      uiState               := 20;
    END_IF
END_CASE
CASE uiState OF
  20:
    stState.bBusy           := FALSE;
    eStateActive            := eState + e_AxisFunction.AXIS_DONE;
    eStateExec	            := e_AxisFunction.AXIS_DONE;

  99:
    stState.bError          := TRUE;
    stState.bBusy           := FALSE;
    eStateActive            := eState + e_AxisFunction.ERROR;
    eStateExec	            := e_AxisFunction.ERROR;
END_CASE
END_ACTION

ACTION Axis_Halt:
CASE uiState OF
  0:
    eStateActive            := eState;
    stState.bBusy           := TRUE;
    stState.bReady          := FALSE;

    stMcOut                 := fbAxis.Halt(Execute        := FALSE,
                                           Deceleration	  := stCtrl.rDec, 
                                           Jerk					  := 100_000.0, 
                                           BufferMode		  := Tc2_MC2.MC_BufferMode.MC_Aborting);
    uiState                 := 10;
END_CASE
CASE uiState OF
  10:
    eStateActive            := eState + e_AxisFunction.AXIS_BUSY;
    eStateExec	            := e_AxisFunction.AXIS_BUSY;

    stMcOut                 := fbAxis.Halt(Execute        := TRUE,
                                           Deceleration	  := stCtrl.rDec, 
                                           Jerk					  := 100_000.0, 
                                           BufferMode		  := Tc2_MC2.MC_BufferMode.MC_Aborting);

    IF NOT stMcOut.Busy
    THEN
      IF stMcOut.Error
      THEN
        stState.uiErrorId		:= stMcOut.ErrorID;

        uiState             := 99;
  
      ELSIF stMcOut.Done
      THEN
        uiState             := 20;
      END_IF
      fbAxis.Halt(Execute         := FALSE,
                  Deceleration	  := stCtrl.rDec, 
                  Jerk					  := 100_000.0, 
                  BufferMode		  := Tc2_MC2.MC_BufferMode.MC_Aborting);
    END_IF
END_CASE
CASE uiState OF
  20:
    stState.bBusy           := FALSE;
    eStateActive            := eState + e_AxisFunction.AXIS_DONE;
    eStateExec		          := e_AxisFunction.AXIS_DONE;

  99:
    stState.bError          := TRUE;
    stState.bBusy           := FALSE;
    eStateActive            := eState + e_AxisFunction.ERROR;
    eStateExec	            := e_AxisFunction.ERROR;
END_CASE
END_ACTION

ACTION Axis_Home:
CASE uiState OF
  0:
    eStateActive            := eState;
    stState.bBusy           := TRUE;

    stMcOut                 := fbAxis.Home(Execute    := FALSE,
                                           Position		:= stHomingOptions.Position, 
                                           HomingMode	:= Tc2_MC2.MC_HomingMode.MC_ResetCalibration, 
                                           Options		:= stHomingOptions.Options);
    IF NOT bXenaxDrive
    THEN
      IF fbAxis.pAxisRef^.Status.Homed
      THEN
        uiState             := 10;
      ELSE
        uiState             := 15;
      END_IF
    ELSE
      uiState               := 100;
    END_IF
END_CASE
CASE uiState OF
  10:
    // always reset calibration to force a homing run of the axis
    eStateActive            := eState + e_AxisFunction.AXIS_BUSY;
    eStateExec	            := e_AxisFunction.AXIS_BUSY;

    stState.bReferenced     := FALSE;

    stMcOut                 := fbAxis.Home(Execute    := TRUE,
                                           Position		:= stHomingOptions.Position, 
                                           HomingMode	:= Tc2_MC2.MC_HomingMode.MC_ResetCalibration, 
                                           Options		:= stHomingOptions.Options);
    IF stMcOut.Done
    THEN
      stMcOut               := fbAxis.Home(Execute    := FALSE,
                                           Position		:= stHomingOptions.Position, 
                                           HomingMode	:= stHomingOptions.HomingMode, 
                                           Options		:= stHomingOptions.Options);

      IF (stHomingOptions.HomingMode = Tc2_MC2.MC_HomingMode.MC_Absolute)
      THEN
        uiState             := 20;
      ELSE
        uiState             := 15;	
      END_IF
    END_IF
END_CASE
CASE uiState OF
  15:
    stMcOut                 := fbAxis.Home(Execute    := TRUE,
                                           Position		:= stHomingOptions.Position, 
                                           HomingMode	:= stHomingOptions.HomingMode, 
                                           Options		:= stHomingOptions.Options);

    IF stMcOut.Done
    THEN
      stState.bReferenced   := fbAxis.pAxisRef^.Status.Homed;

      stMcOut               := fbAxis.Home(Execute    := FALSE,
                                           Position		:= stHomingOptions.Position, 
                                           HomingMode	:= stHomingOptions.HomingMode, 
                                           Options		:= stHomingOptions.Options);
      uiState               := 20;

    ELSIF stMcOut.Error
    THEN
      stState.uiErrorId		  := stMcOut.ErrorID;
      stMcOut               := fbAxis.Home(Execute    := FALSE,
                                           Position		:= stHomingOptions.Position, 
                                           HomingMode	:= stHomingOptions.HomingMode, 
                                           Options		:= stHomingOptions.Options);
      uiState               := 99;
    END_IF

  20:
    stState.bBusy           := FALSE;
    eStateActive            := eState + e_AxisFunction.AXIS_DONE;
    eStateExec	            := e_AxisFunction.AXIS_DONE;

  99:
    stState.bError          := TRUE;
    stState.bBusy           := FALSE;
    eStateActive            := eState + e_AxisFunction.ERROR;
    eStateExec	            := e_AxisFunction.ERROR;
END_CASE
CASE uiState OF
  // Xenax drive homing
  100:
    eStateActive            := eState + e_AxisFunction.AXIS_BUSY;
    stState.bReferenced 		:= FALSE;
    fbXenaxHoming.bExecute 	:= FALSE;

    uiState                 := 110;
END_CASE
CASE uiState OF
  110:
    fbXenaxHoming.bExecute  := TRUE;
    uiState                 := 120;

  120:
    IF fbXenaxHoming.Error
    THEN
      stState.uiErrorId     := fbXenaxHoming.ErrorId;
      uiState               := 99;

    ELSIF fbXenaxHoming.Done
    THEN
      stState.bReferenced 	:= TRUE;
      fbXenaxHoming.bExecute:= FALSE;

      uiState               := 20;
    END_IF
END_CASE
END_ACTION

ACTION Axis_Idle:
IF stState.bReady
THEN
  IF NOT fbAxis.pAxisRef^.Status.Error
  THEN
    stState.bError  := FALSE;
  END_IF
  eStateActive      := eState;
  eStateExec	      := e_AxisFunction.AXIS_DONE;
END_IF

IF NOT stState.bReady
THEN
  eStateActive := eState;
  eStateExec	 := e_AxisFunction.AXIS_BUSY;
END_IF
END_ACTION

ACTION Axis_Init:
(*
-------------------------------------------------------------------------------
	INIT 
  - check for fbAxis to startUp --> sAxisName chec
  - check for fbAxis StartUpError --> Axis_Reset() and try again

  - get encodertype and set output bSercosAxis
	- get Axis Params from NC
	- get manufacturer device name for detecting use of Xenax drive

-------------------------------------------------------------------------------
*)
CASE uiInitState OF

  0:
  stState.bError          := FALSE;
  isizeOut                := SIZEOF(stState);
  iSizeIn	                := SIZEOF(stCtrl);
  bSercosAxis             := FALSE;
  sAxisName               := fbAxis.NcAxisName;

  IF fbAxis.StartUpDone
  THEN
    stMsg.eType 				  := E_MessageType.eMessageInfo;
    stMsg.eDevice 			  := E_Device.Axis;
    stMsg.eSubdevice 		  := e_Subdevice.General;
    stMsg.iErrorNumber 	  := fbAxis.pAxisRef^.NcToPlc.AxisId;
    stMsg.sText					  := 'Init: ';
    stMsg.sText					  := Tc2_Standard.CONCAT(stMsg.sText, sAxisName);
    f_MessageSet(stMsg);

    uiInitState           := 40;
    bXenaxDrive				    := FALSE;
    bSercosAxis           := FALSE;

    fbCoeRead(Execute	    := FALSE,
              NetId       := fbAxis.pAxisRef^.ADS.NetId, 
              Axis        := fbAxis.pAxisRef^);

    IF (fbAxis.EncoderType <> 1)
    THEN
      uiInitState         := 10;
    END_IF

  ELSE
    IF (stMsg.sText <> 'startup')
    THEN
      stMsg.eType 				:= E_MessageType.eMessageInfo;
      stMsg.eDevice 			:= E_Device.Axis;
      stMsg.eSubdevice 		:= e_Subdevice.General;
      stMsg.iErrorNumber 	:= fbAxis.pAxisRef^.NcToPlc.AxisId;
      stMsg.sText					:= 'startup';
      f_MessageSet(stMsg);
    END_IF

    IF (fbAxis.StartUpError)
    THEN
      stMsg.eType 				:= E_MessageType.eMessageError;
      stMsg.eDevice 			:= E_Device.Axis;
      stMsg.eSubdevice 		:= e_Subdevice.General;
      stMsg.iErrorNumber 	:= fbAxis.pAxisRef^.NcToPlc.AxisId;
      stMsg.sText					:= 'InitError: ';

      f_MessageSet(stMsg);

      uiInitState         := 90;
    END_IF
  END_IF

  10:
    // get manufacturer device name in CoE
    fbCoeRead.Index 		  := 16#1008;
    fbCoeRead.SubIndex 	  := 0;
    fbCoeRead.pDstBuf		  := ADR(sDriveType);
    fbCoeRead.BufLen		  := SIZEOF(sDriveType);

    fbCoeRead(Execute	    := TRUE,
              NetId       := fbAxis.pAxisRef^.ADS.NetId, 
              Axis        := fbAxis.pAxisRef^);

    IF fbCoeRead.Busy
    THEN
      uiInitState         := 20;
    END_IF

  20:
    fbCoeRead(
              NetId       := fbAxis.pAxisRef^.ADS.NetId, 
              Axis        := fbAxis.pAxisRef^);

    IF (fbCoeRead.Error)
    THEN
      uiInitState         := 90;

    ELSIF NOT fbCoeRead.Busy
    THEN
      stState.bError 		  := FALSE;
      stState.uiErrorId   := 0;
      uiInitState         := 30;
    END_IF

  30:
    IF (fbAxis.EncoderType = 8) OR
       (fbAxis.EncoderType = 9)
    THEN
      bSercosAxis         := TRUE;

      stMsg.eType 				:= E_MessageType.eMessageInfo;
      stMsg.eDevice 			:= E_Device.Axis;
      stMsg.eSubdevice 		:= e_Subdevice.General;
      stMsg.iErrorNumber 	:= fbAxis.pAxisRef^.NcToPlc.AxisId;
      stMsg.sText					:= Tc2_Standard.CONCAT(stMsg.sText,',');
      stMsg.sText					:= Tc2_Standard.CONCAT(stMsg.sText, 'SERCOS');
      f_MessageSet(stMsg);
    END_IF

    // check manufacturer device name for identifier string
    IF (FIND(sDriveType, sXenax) <> 0)
    THEN
      bXenaxDrive         := TRUE;

      stMsg.eType 				:= E_MessageType.eMessageInfo;
      stMsg.eDevice 			:= E_Device.Axis;
      stMsg.eSubdevice 		:= e_Subdevice.General;
      stMsg.iErrorNumber 	:= fbAxis.pAxisRef^.NcToPlc.AxisId;
      stMsg.sText					:= Tc2_Standard.CONCAT(stMsg.sText,',');
      stMsg.sText					:= Tc2_Standard.CONCAT(stMsg.sText,sXenax);
      f_MessageSet(stMsg);
    END_IF
    uiInitState           := 40;

  40:
    eStateExec	          := e_AxisFunction.AXIS_DONE;
    eStateExecOld         := e_AxisFunction.AXIS_DONE;
    stMsg.eType 				  := E_MessageType.eMessageInfo;
    stMsg.eDevice 			  := E_Device.Axis;
    stMsg.eSubdevice 		  := e_Subdevice.General;
    stMsg.iErrorNumber 	  := fbAxis.pAxisRef^.NcToPlc.AxisId;
    stMsg.sText					  := Tc2_Standard.CONCAT(stMsg.sText, ': ');
    stMsg.sText					  := Tc2_Standard.CONCAT(stMsg.sText, TO_STRING(eStateExec));
    f_MessageSet(stMsg);
    uiInitState           := 100;

  90:
    stState.bError        := TRUE;
    uiState               := 0;
    uiInitState           := 91;

  91:
    Axis_Reset();
    IF (eStateExec = e_AxisFunction.AXIS_DONE)
    THEN
      stMsg.eType 				:= E_MessageType.eMessageInfo;
      stMsg.eDevice 			:= E_Device.Axis;
      stMsg.eSubdevice 		:= e_Subdevice.General;
      stMsg.iErrorNumber 	:= fbAxis.pAxisRef^.NcToPlc.AxisId;
      stMsg.sText					:= 'Init Axis_Reset: ';

      uiInitState         := 0;
    END_IF

  100:
    bInit                 := TRUE;
END_CASE
END_ACTION

ACTION Axis_Move_Buffer:
CASE uiState OF
  0:
    eStateActive            := eState;
    stState.bBusy           := TRUE;
    stState.bReady          := FALSE;

    stMcOut                 := fbAxis.MoveAbsolute(Enable       := FALSE,
                                                   Position		  := stCtrl.rSetPos, 
                                                   Velocity		  := stCtrl.rSetVelo, 
                                                   Acceleration := stCtrl.rAcc, 
                                                   Deceleration := stCtrl.rDec, 
                                                   Jerk				  := 0, 
                                                   BufferMode	      := stMotionOptions.eBufferMode,
                                                   fActivePosition  := stState.rSetPos,
                                                   eState           := eBufferState);

    uiState                 := 10;
END_CASE
CASE uiState OF
  10:
    eStateActive            := eState + e_AxisFunction.AXIS_BUSY;
    eStateExec              := e_AxisFunction.AXIS_BUSY;

    stMcOut                 := fbAxis.MoveAbsolute(Enable       := TRUE,
                                                   Position     := stCtrl.rSetPos, 
                                                   Velocity     := stCtrl.rSetVelo, 
                                                   Acceleration := stCtrl.rAcc, 
                                                   Deceleration := stCtrl.rDec, 
                                                   Jerk         := 0, 
                                                   BufferMode	      := stMotionOptions.eBufferMode,
                                                   fActivePosition  := stState.rSetPos,
                                                   eState           := eBufferState);

    IF stMcOut.Error
    THEN
      stState.uiErrorId     := stMcOut.ErrorID;
      uiState               := 99;

      stMcOut               := fbAxis.MoveAbsolute(Enable     := FALSE,
                                                   Position		  := stCtrl.rSetPos, 
                                                   Velocity		  := stCtrl.rSetVelo, 
                                                   Acceleration := stCtrl.rAcc, 
                                                   Deceleration := stCtrl.rDec, 
                                                   Jerk				  := 0, 
                                                   BufferMode	      := stMotionOptions.eBufferMode,
                                                   fActivePosition  := stState.rSetPos,
                                                   eState           := eBufferState);

    END_IF
END_CASE
CASE uiState OF
  99:
    stState.bError          := TRUE;
    stState.bBusy           := FALSE;
    eStateActive            := eState + e_AxisFunction.ERROR;
    eBufferState            :=
    eStateExec	            := e_AxisFunction.ERROR;
END_CASE
END_ACTION

ACTION Axis_Move_Buffer_Velocity:
CASE uiState OF
  0:
    eStateActive            := eState;
    stState.bBusy           := TRUE;
    stState.bReady          := FALSE;
    uiState                 := 5;
END_CASE

CASE uiState OF
  5:
    eStateActive            := eState + e_AxisFunction.AXIS_BUSY;
    eStateExec	            := e_AxisFunction.AXIS_BUSY;

    stMcOut                 := fbAxis.MoveVelocity(FALSE,
                                                   stCtrl.rSetVelo,
                                                   stCtrl.rAcc,
                                                   stCtrl.rDec,
                                                   100_000,
                                                   stCtrl.iDirection,
                                                   BufferMode       := Tc2_MC2.MC_BufferMode.MC_Aborting,
                                                   fActiveVelocity  := stState.rSetPos,
                                                   eState           := eBufferState);
    uiState                 := 10;
END_CASE
CASE uiState OF
  10:
    eStateActive            := eState + e_AxisFunction.AXIS_BUSY;
    eStateExec	            := e_AxisFunction.AXIS_BUSY;

    stMcOut                 := fbAxis.MoveVelocity(TRUE,
                                                   stCtrl.rSetVelo,
                                                   stCtrl.rAcc,
                                                   stCtrl.rDec,
                                                   100_000,
                                                   stCtrl.iDirection,
                                                   BufferMode       := Tc2_MC2.MC_BufferMode.MC_Aborting,
                                                   fActiveVelocity  := stState.rSetPos,
                                                   eState           := eBufferState);

    IF stMcOut.Error
    THEN
      stMcOut               := fbAxis.MoveVelocity(FALSE,
                                                   stCtrl.rSetVelo,
                                                   stCtrl.rAcc,
                                                   stCtrl.rDec,
                                                   100_000,
                                                   stCtrl.iDirection,
                                                   BufferMode       := Tc2_MC2.MC_BufferMode.MC_Aborting,
                                                   fActiveVelocity  := stState.rSetPos,
                                                   eState           := eBufferState);

      stState.uiErrorId		  := stMcOut.ErrorID;

      uiState               := 99;
    END_IF
END_CASE

CASE uiState OF
  99:
    stState.bError          := TRUE;
    stState.bBusy           := FALSE;
    eStateActive            := eState + e_AxisFunction.ERROR;
    eBufferState            :=
    eStateExec	            := e_AxisFunction.ERROR;
END_CASE
END_ACTION

ACTION Axis_Move_Pos:
CASE uiState OF
  0:
    eStateActive            := eState;
    stState.bBusy           := TRUE;

    rSetPos                 := stCtrl.rSetPos;
    stMcOut                 := fbAxis.MovePtP(Execute     := FALSE,
                                              Position		:= rSetPos, 
                                              Velocity		:= stCtrl.rSetVelo, 
                                              Acceleration:= stCtrl.rAcc, 
                                              Deceleration:= stCtrl.rDec, 
                                              Jerk				:= 0);

    uiState                 := 10;
END_CASE
CASE uiState OF
  10:
    eStateActive            := eState + e_AxisFunction.AXIS_BUSY;
    eStateExec	            := e_AxisFunction.AXIS_BUSY;

    stMcOut                 := fbAxis.MovePtP(Execute     := TRUE,
                                              Position		:= rSetPos, 
                                              Velocity		:= stCtrl.rSetVelo, 
                                              Acceleration:= stCtrl.rAcc, 
                                              Deceleration:= stCtrl.rDec, 
                                              Jerk				:= 0); //default

    IF stMcOut.Done OR 
       stMcOut.Error
    THEN
      IF stMcOut.Done
      THEN
        uiState             := 11;
      END_IF
      IF stMcOut.Error
      THEN
        stState.uiErrorId		:= stMcOut.ErrorID;
        uiState             := 99;
      END_IF

      stMcOut               := fbAxis.MovePtP(Execute     := FALSE,
                                              Position		:= rSetPos, 
                                              Velocity		:= stCtrl.rSetVelo, 
                                              Acceleration:= stCtrl.rAcc, 
                                              Deceleration:= stCtrl.rDec, 
                                              Jerk				:= 0);
    END_IF
END_CASE
CASE uiState OF
  11:
    IF stState.bInTarget
    THEN
      uiState               := 20;
    END_IF
END_CASE
CASE uiState OF
  20:
    stState.bBusy           := FALSE;
    eStateActive            := eState + e_AxisFunction.AXIS_DONE;
    eStateExec	            := e_AxisFunction.AXIS_DONE;

  99:
    stState.bError          := TRUE;
    stState.bBusy           := FALSE;
    eStateActive            := eState + e_AxisFunction.ERROR;
    eStateExec              := e_AxisFunction.ERROR;
END_CASE
END_ACTION

ACTION Axis_Move_Velo:
CASE uiState OF
  0:
    eStateActive            := eState;
    stState.bBusy           := TRUE;
    stState.bReady          := FALSE;
    uiState := 5;
END_CASE

CASE uiState OF
  5:
    eStateActive            := eState + e_AxisFunction.AXIS_BUSY;
    eStateExec	            := e_AxisFunction.AXIS_BUSY;

    stMcOut                 := fbAxis.MoveVelocity(FALSE,
                                                   stCtrl.rSetVelo,
                                                   stCtrl.rAcc,
                                                   stCtrl.rDec,
                                                   100_000,
                                                   stCtrl.iDirection,
                                                   BufferMode       := Tc2_MC2.MC_BufferMode.MC_Aborting,
                                                   fActiveVelocity  := stState.rSetPos,
                                                   eState           := eBufferState);

    uiState                 := 10;
END_CASE
CASE uiState OF
  10:
    eStateActive            := eState + e_AxisFunction.AXIS_BUSY;
    eStateExec	            := e_AxisFunction.AXIS_BUSY;

    stMcOut                 := fbAxis.MoveVelocity(TRUE,
                                                   stCtrl.rSetVelo,
                                                   stCtrl.rAcc,
                                                   stCtrl.rDec,
                                                   100_000,
                                                   stCtrl.iDirection,
                                                   BufferMode       := Tc2_MC2.MC_BufferMode.MC_Aborting,
                                                   fActiveVelocity  := stState.rSetPos,
                                                   eState           := eBufferState);

    IF stMcOut.Error
    THEN
      stMcOut               := fbAxis.MoveVelocity(FALSE,
                                                   stCtrl.rSetVelo,
                                                   stCtrl.rAcc,
                                                   stCtrl.rDec,
                                                   100_000,
                                                   stCtrl.iDirection,
                                                   BufferMode       := Tc2_MC2.MC_BufferMode.MC_Aborting,
                                                   fActiveVelocity  := stState.rSetPos,
                                                   eState           := eBufferState);

      stState.uiErrorId     := stMcOut.ErrorID;

      uiState               := 99;

    ELSIF stMcOut.Done
    THEN
      stMcOut               := fbAxis.MoveVelocity(FALSE,
                                                   stCtrl.rSetVelo,
                                                   stCtrl.rAcc,
                                                   stCtrl.rDec,
                                                   100_000,
                                                   stCtrl.iDirection,
                                                   BufferMode       := Tc2_MC2.MC_BufferMode.MC_Aborting,
                                                   fActiveVelocity  := stState.rSetPos,
                                                   eState           := eBufferState);

      uiState               := 20;
    END_IF
END_CASE

CASE uiState OF
  20:
    stState.bBusy           := FALSE;
    eStateActive            := eState + e_AxisFunction.AXIS_DONE;
    eStateExec              := e_AxisFunction.AXIS_DONE;

  99:
    stState.bError          := TRUE;
    stState.bBusy           := FALSE;
    eStateActive            := eState + e_AxisFunction.ERROR;
    eStateExec              := e_AxisFunction.ERROR;
END_CASE
END_ACTION

ACTION Axis_Parameter:
CASE uiState OF
  0:
    eStateActive            := eState;

    tonWaitSeq(IN           := FALSE);

    IF stNcParameter.bRead
    THEN
      stState.bBusy         := TRUE;
      stMcOut               := fbAxis.ReadParameter(FALSE,stNcParameter.ParameterNumber);
      uiState               := 10;

    ELSIF stNcParameter.bWrite
    THEN
      stState.bBusy         := TRUE;
      stMcOut               := fbAxis.WriteParameter(FALSE, stNcParameter.ParameterNumber, stNcParameter.rValueWrite);
      uiState               := 11;
    END_IF

  10:
    eStateActive            := eState + e_AxisFunction.AXIS_BUSY;
    eStateExec              := e_AxisFunction.AXIS_BUSY;

    tonWaitSeq(IN           := TRUE, 
               PT           := T#50MS);

    stMcOut                 := fbAxis.ReadParameter(TRUE,stNcParameter.ParameterNumber);

    IF stMcOut.Done AND 
       tonWaitSeq.Q
    THEN
      stNcParameter.rValueRead  := LREAL_TO_REAL(fbAxis.ReadParamValue);
      stMcOut                   := fbAxis.ReadParameter(FALSE,stNcParameter.ParameterNumber);

      uiState               := 20;
    END_IF

  11:
    eStateActive            := eState + e_AxisFunction.AXIS_BUSY;
    eStateExec              := e_AxisFunction.AXIS_BUSY;

    tonWaitSeq(IN           := TRUE, 
               PT           := T#50MS);

    stMcOut                 := fbAxis.WriteParameter(TRUE, stNcParameter.ParameterNumber, stNcParameter.rValueWrite);

    IF stMcOut.Done AND 
       tonWaitSeq.Q
    THEN
      IF fbAxis.LocalParameterReload()
      THEN
        stMcOut             := fbAxis.WriteParameter(FALSE, stNcParameter.ParameterNumber, stNcParameter.rValueWrite);
        uiState             := 20;
      END_IF
    END_IF

  20:
    stState.bBusy           := FALSE;
    eStateActive            := eState + e_AxisFunction.AXIS_DONE;
    eStateExec              := e_AxisFunction.AXIS_DONE;
END_CASE
END_ACTION

ACTION Axis_Reset:
CASE uiState OF
  0:
    eStateActive            := eState;
    stState.bBusy           := TRUE;
    stState.bReady          := FALSE;
    stState.bTimeout        := FALSE;
    stMcOut                 := fbAxis.ErrorReset(FALSE);

    uiState                 := 10;
END_CASE
CASE uiState OF
  10:
    eStateActive            := eState + e_AxisFunction.AXIS_BUSY;
    eStateExec              := e_AxisFunction.AXIS_BUSY;
    stMcOut                 := fbAxis.ErrorReset(TRUE);

    IF stMcOut.Done
    THEN
      stState.bError        := FALSE;
      stState.uiErrorId     := 0;
      stMcOut               := fbAxis.ErrorReset(FALSE);
      uiState               := 20;

    ELSIF stMcOut.Error
    THEN
      stState.uiErrorId		  := stMcOut.ErrorID;
      uiState               := 99;
    END_IF
END_CASE
CASE uiState OF
  20:
    fbResetSercos(bExecute	:= FALSE);

    IF fbAxis.pAxisRef^.Status.DriveDeviceError AND
       bSercosAxis
    THEN
      tonTimeout(IN         := FALSE, 
                 PT         := tUpdate);

      uiState               := 30;
    ELSE
      uiState               := 40;
    END_IF

END_CASE
CASE uiState OF
  30:
    tonTimeout(IN           := TRUE, 
               PT           := tUpdate);

    fbResetSercos(bExecute	:= TRUE, 
                  p_AxisRef	:= ADR(fbAxis._AxisRef), stMcOutput=> );

    IF tonTimeout.Q
    THEN
      uiState               := 0;
    ELSE
      IF NOT fbAxis.pAxisRef^.Status.DriveDeviceError
      THEN
        tonTimeout(IN       := FALSE, 
                   PT       := tUpdate);

        uiState             := 40;
      END_IF
    END_IF
END_CASE
CASE uiState OF
  40:
    stState.bBusy           := FALSE;
    eStateActive            := eState + e_AxisFunction.AXIS_DONE;
    eStateExec              := e_AxisFunction.AXIS_DONE;


  99:
    stState.bError          := TRUE;
    stState.bBusy           := FALSE;
    eStateActive            := eState + e_AxisFunction.ERROR;
    eStateExec              := e_AxisFunction.ERROR;
END_CASE
END_ACTION

ACTION Axis_Reset_SS1:
CASE uiState OF
  0:
    eStateActive            := eState;
    stState.bBusy           := TRUE;
    stState.bReady          := FALSE;
    stState.bTimeout        := FALSE;
    stMcOut                 := fbAxis.ErrorReset(FALSE);

    uiState                 := 10;
END_CASE
CASE uiState OF
  10:
    eStateActive            := eState + e_AxisFunction.AXIS_BUSY;
    eStateExec              := e_AxisFunction.AXIS_BUSY;
    stMcOut                 := fbAxis.ErrorReset(TRUE);

    IF NOT stMcOut.Busy
    THEN
      stMcOut               := fbAxis.ErrorReset(FALSE);
      uiState               := 20;

    ELSIF stMcOut.Error
    THEN
      stState.uiErrorId		  := stMcOut.ErrorID;
      uiState               := 99;
    END_IF
END_CASE
CASE uiState OF
  20:
    fbResetSercos(bExecute	:= FALSE);

    IF fbAxis.pAxisRef^.Status.DriveDeviceError AND
       bSercosAxis
    THEN
      tonTimeout(IN         := FALSE, 
                 PT         := tUpdate);

      uiState               := 30;
    ELSE
      uiState               := 40;
    END_IF

END_CASE
CASE uiState OF
  30:
    tonTimeout(IN           := TRUE, 
               PT           := tUpdate);

    fbResetSercos(bExecute	:= TRUE, 
                  p_AxisRef	:= ADR(fbAxis._AxisRef), stMcOutput=> );

    IF tonTimeout.Q
    THEN
      uiState               := 0;
    ELSE
      IF NOT fbAxis.pAxisRef^.Status.DriveDeviceError
      THEN
        tonTimeout(IN       := FALSE, 
                   PT       := tUpdate);

        uiState             := 40;
      END_IF
    END_IF
END_CASE
CASE uiState OF
  40:
    stState.bBusy           := FALSE;
    eStateActive            := eState + e_AxisFunction.AXIS_DONE;
    eStateExec              := e_AxisFunction.AXIS_DONE;


  99:
    stState.bError          := TRUE;
    stState.bBusy           := FALSE;
    eStateActive            := eState + e_AxisFunction.ERROR;
    eStateExec              := e_AxisFunction.ERROR;
END_CASE
END_ACTION

ACTION Axis_Stop:
CASE uiState OF
  0:
    eStateActive            := eState;
    stState.bBusy           := TRUE;
    stState.bReady          := FALSE;

    stMcOut                 := fbAxis.Stop(FALSE);
    uiState                 := 10;
END_CASE
CASE uiState OF
  10:
    eStateActive            := eState + e_AxisFunction.AXIS_BUSY;
    eStateExec              := e_AxisFunction.AXIS_BUSY;

    stMcOut                 := fbAxis.Stop(TRUE);

    IF stMcOut.Error
    THEN
      stState.uiErrorId		  := stMcOut.ErrorID;
      stMcOut               := fbAxis.Stop(FALSE);
      uiState               := 99;

    ELSIF stMcOut.Done
    THEN
      stMcOut               := fbAxis.Stop(FALSE);
      uiState               := 20;
    END_IF
END_CASE
CASE uiState OF
  20:
    stState.bBusy           := FALSE;

    eStateActive            := eState + e_AxisFunction.AXIS_DONE;
    eStateExec              := e_AxisFunction.AXIS_DONE;

  99:
    stState.bError          := TRUE;
    stState.bBusy           := FALSE;

    eStateActive            := eState + e_AxisFunction.ERROR;
    eStateExec              := e_AxisFunction.ERROR;
END_CASE
END_ACTION

ACTION Axis_Stop_SS1:

eStateActive                := e_AxisFunction.AXIS_SS1_STOP + e_AxisFunction.AXIS_BUSY;
eStateExec	                := e_AxisFunction.AXIS_BUSY;

stState.bBusy               := TRUE;
stState.bReady              := FALSE;

CASE uiStateSS1 OF
   0:
    IF fbAxis.Enable
    THEN
      uiStateSS1            := 10;
    ELSE
      uiStateSS1            := 100;
    END_IF
END_CASE
CASE uiStateSS1 OF
  10:
    fbAxis.Stop(FALSE);
    uiStateSS1              := 20;
END_CASE
CASE uiStateSS1 OF
  20:
    fbAxis.Stop(TRUE);
    IF fbAxis._AxisRef.Status.NotMoving
    THEN
      uiStateSS1            := 100;
    END_IF
END_CASE
CASE uiStateSS1 OF
  100:
    uiStateSS1              := 0;
    fbAxis.Enable           := FALSE;
    stState.bBusy           := FALSE;
    eStateActive            := e_AxisFunction.AXIS_SS1_STOP + e_AxisFunction.AXIS_DONE;
    eStateExec              := e_AxisFunction.AXIS_DONE;
END_CASE
END_ACTION

ACTION Axis_WriteBufferMode:

CASE uiState OF
  0:
    eStateActive            := eState;
    stState.bBusy           := TRUE;
    stState.bReady          := FALSE;

    uiState                 := 10;
END_CASE
CASE uiState OF
  10:
    eStateActive            := eState + e_AxisFunction.AXIS_BUSY;
    eStateExec	            := e_AxisFunction.AXIS_BUSY;

END_CASE
CASE uiState OF
  20:
    stState.bBusy           := FALSE;
    eStateActive            := eState + e_AxisFunction.AXIS_DONE;
    eStateExec	            := e_AxisFunction.AXIS_DONE;

  99:
    stState.bError          := TRUE;
    stState.bBusy           := FALSE;
    eStateActive            := eState + e_AxisFunction.ERROR;
    eStateExec	            := e_AxisFunction.ERROR;
END_CASE
END_ACTION

PROPERTY MasterAxis1 : POINTER TO Tc2_MC2.AXIS_REF
GET
MasterAxis1 := _pAxis1;
END_GET
SET
IF MasterAxis1 = 0 THEN
	_pAxis1 := ADR(st_AxisREF_Dummy);
ELSE
	_pAxis1 := MasterAxis1;	
END_IF
END_SET
END_PROPERTY

PROPERTY MasterAxis2 : POINTER TO Tc2_MC2.AXIS_REF
GET
MasterAxis2 := _pAxis2;
END_GET
SET
IF MasterAxis2 = 0 THEN
	_pAxis2 := ADR(st_AxisREF_Dummy);
ELSE
	_pAxis2 := MasterAxis2;	
END_IF
END_SET
END_PROPERTY

PROPERTY MasterAxis3 : POINTER TO Tc2_MC2.AXIS_REF
GET
MasterAxis3 := _pAxis3;
END_GET
SET
IF MasterAxis3 = 0 THEN
	_pAxis3 := ADR(st_AxisREF_Dummy);
ELSE
	_pAxis3 := MasterAxis3;	
END_IF
END_SET
END_PROPERTY

PROPERTY MasterAxis4 : POINTER TO Tc2_MC2.AXIS_REF
GET
MasterAxis4 := _pAxis4;
END_GET
SET
IF MasterAxis4 = 0 THEN
	_pAxis4 := ADR(st_AxisREF_Dummy);
ELSE
	_pAxis4 := MasterAxis4;	
END_IF
END_SET
END_PROPERTY

PROPERTY PUBLIC StatusCompact : ST_AxisStatusCompact
GET


_stStatusCompact.Error                := fbAxis.pAxisRef^.Status.Error;
(* PLCopen motion control statemachine states: *)
_stStatusCompact.ErrorStop            := fbAxis.pAxisRef^.Status.ErrorStop;
_stStatusCompact.Disabled             := fbAxis.pAxisRef^.Status.Disabled;
_stStatusCompact.Stopping             := fbAxis.pAxisRef^.Status.Stopping;

_stStatusCompact.StandStill           := fbAxis.pAxisRef^.Status.StandStill;
_stStatusCompact.DiscreteMotion       := fbAxis.pAxisRef^.Status.DiscreteMotion;
_stStatusCompact.ContinuousMotion     := fbAxis.pAxisRef^.Status.ContinuousMotion; 
_stStatusCompact.SynchronizedMotion   := fbAxis.pAxisRef^.Status.SynchronizedMotion;

_stStatusCompact.Homing               := fbAxis.pAxisRef^.Status.Homing;

(* additional status - (PLCopen definition)*)
_stStatusCompact.ConstantVelocity     := fbAxis.pAxisRef^.Status.ConstantVelocity; 
_stStatusCompact.Accelerating         := fbAxis.pAxisRef^.Status.Accelerating;
_stStatusCompact.Decelerating         := fbAxis.pAxisRef^.Status.Decelerating;

(* Axis.NcToPlc.StateDWord *)
_stStatusCompact.Operational          := fbAxis.pAxisRef^.Status.Operational; 
_stStatusCompact.ControlLoopClosed    := fbAxis.pAxisRef^.Status.ControlLoopClosed;
_stStatusCompact.HasJob               := fbAxis.pAxisRef^.Status.HasJob; 
_stStatusCompact.HasBeenStopped       := fbAxis.pAxisRef^.Status.HasBeenStopped; 
_stStatusCompact.NewTargetPosition    := fbAxis.pAxisRef^.Status.NewTargetPosition;
_stStatusCompact.InPositionArea       := fbAxis.pAxisRef^.Status.InPositionArea; 
_stStatusCompact.InTargetPosition     := fbAxis.pAxisRef^.Status.InTargetPosition; 

_stStatusCompact.Homed                := fbAxis.pAxisRef^.Status.Homed; 
_stStatusCompact.HomingBusy           := fbAxis.pAxisRef^.Status.HomingBusy; 
_stStatusCompact.MotionCommandsLocked := fbAxis.pAxisRef^.Status.MotionCommandsLocked;
_stStatusCompact.SoftLimitMinExceeded := fbAxis.pAxisRef^.Status.SoftLimitMinExceeded;
_stStatusCompact.SoftLimitMaxExceeded := fbAxis.pAxisRef^.Status.SoftLimitMaxExceeded;

_stStatusCompact.Moving               := fbAxis.pAxisRef^.Status.Moving; 
_stStatusCompact.PositiveDirection    := fbAxis.pAxisRef^.Status.PositiveDirection; 
_stStatusCompact.NegativeDirection    := fbAxis.pAxisRef^.Status.NegativeDirection; 
_stStatusCompact.NotMoving            := fbAxis.pAxisRef^.Status.NotMoving; 
_stStatusCompact.Compensating         := fbAxis.pAxisRef^.Status.Compensating;

_stStatusCompact.ExtSetPointGenEnabled:= fbAxis.pAxisRef^.Status.ExtSetPointGenEnabled; 
_stStatusCompact.ExternalLatchValid   := fbAxis.pAxisRef^.Status.ExternalLatchValid; 
_stStatusCompact.CamDataQueued        := fbAxis.pAxisRef^.Status.CamDataQueued; 
_stStatusCompact.CamTableQueued       := fbAxis.pAxisRef^.Status.CamTableQueued; 
_stStatusCompact.CamScalingPending    := fbAxis.pAxisRef^.Status.CamScalingPending; 
_stStatusCompact.CmdBuffered          := fbAxis.pAxisRef^.Status.CmdBuffered; 
_stStatusCompact.PTPmode              := fbAxis.pAxisRef^.Status.PTPmode; 
_stStatusCompact.DriveDeviceError     := fbAxis.pAxisRef^.Status.DriveDeviceError; 
_stStatusCompact.IoDataInvalid        := fbAxis.pAxisRef^.Status.IoDataInvalid; 

(* Axis.NcToPlc.CoupleState *)
_stStatusCompact.Coupled              := fbAxis.pAxisRef^.Status.Coupled;

StatusCompact := _stStatusCompact;
END_GET
END_PROPERTY

PROPERTY stCam : ST_CamIn
GET
stCam := _stCamIn;
END_GET
SET
_stCamIn := stCam;

IF NOT IsFinite(F_Real(_stCamIn.MasterOffset))
THEN
  _stCamIn.MasterOffset := 0.0;
END_IF

IF NOT IsFinite(F_Real(_stCamIn.SlaveOffset))
THEN
  _stCamIn.SlaveOffset := 0.0;
END_IF

IF NOT IsFinite(F_Real(_stCamIn.MasterScaling))
THEN
  _stCamIn.MasterScaling := 0.0;
END_IF

IF NOT IsFinite(F_Real(_stCamIn.SlaveScaling))
THEN
  _stCamIn.SlaveScaling := 0.0;
END_IF
END_SET
END_PROPERTY

PROPERTY stGear : ST_GearIn
GET
stGear := _stGearIn;
END_GET
SET
_stGearIn := stGear;

IF NOT IsFinite(F_Real(_stGearIn.Acceleration))
THEN
  _stGearIn.Acceleration := 0.0;
END_IF

IF NOT IsFinite(F_Real(_stGearIn.Deceleration))
THEN
  _stGearIn.Deceleration := 0.0;
END_IF

IF NOT IsFinite(F_Real(_stGearIn.Jerk))
THEN
  _stGearIn.Jerk := 0.0;
END_IF

IF NOT IsFinite(F_Real(_stGearIn.RatioNumerator))
THEN
  _stGearIn.RatioNumerator := 0.0;
END_IF
END_SET
END_PROPERTY

PROPERTY stGearMultiMaster : ST_GearInMultiMaster
GET
stGearMultiMaster := _stGearInMultiMaster;
END_GET
SET
_stGearInMultiMaster := stGearMultiMaster;

IF NOT IsFinite(F_Real(_stGearInMultiMaster.Acceleration))
THEN
  _stGearInMultiMaster.Acceleration := 0.0;
END_IF

IF NOT IsFinite(F_Real(_stGearInMultiMaster.Deceleration))
THEN
  _stGearInMultiMaster.Deceleration := 0.0;
END_IF

IF NOT IsFinite(F_Real(_stGearInMultiMaster.Jerk))
THEN
  _stGearInMultiMaster.Jerk := 0.0;
END_IF

IF NOT IsFinite(F_Real(_stGearInMultiMaster.GearRatio1))
THEN
  _stGearInMultiMaster.GearRatio1 := 0.0;
END_IF

IF NOT IsFinite(F_Real(_stGearInMultiMaster.GearRatio2))
THEN
  _stGearInMultiMaster.GearRatio2 := 0.0;
END_IF

IF NOT IsFinite(F_Real(_stGearInMultiMaster.GearRatio3))
THEN
  _stGearInMultiMaster.GearRatio3 := 0.0;
END_IF

IF NOT IsFinite(F_Real(_stGearInMultiMaster.GearRatio4))
THEN
  _stGearInMultiMaster.GearRatio4 := 0.0;
END_IF
END_SET
END_PROPERTY

END_FUNCTION_BLOCK

// ---- POUs/NC_AXIS/FB_McPtpAxis.TcPOU
FUNCTION_BLOCK FB_McPtpAxis IMPLEMENTS I_McAxis
VAR
  _AxisRef                    : Tc2_MC2.AXIS_REF;
  pCalibrationCam             : POINTER TO BOOL;
  bConnectProps2NcParams      : BOOL := TRUE;
  stDefaultAcceleration       : ST_Param;
  stDefaultDeceleration       : ST_Param;
  stDefaultJerk               : ST_Param;
  fDefaultVelocity            : LREAL;

  stHomingSearchVelo          : ST_Param;
  stHomingVelo                : ST_Param;
  stMaxAcceleration           : ST_Param;
  stMaxDeceleration           : ST_Param;
  stMaxVelocity               : ST_Param;
  stTargetPositionWindow      : ST_Param;


  stSwPosLimitNegative        : ST_Param;
  stSwPosLimitNegativeActive  : ST_BoolParam;
  stSwPosLimitPositive        : ST_Param;
  stSwPosLimitPositiveActive  : ST_BoolParam;
  fReadParamValue             : LREAL;
  stAxisStatus                : Tc2_MC2.ST_AxisStatus;

  // name and encoder type are read by ADSREAD instance from NC
  stAxisName                  : STRING(30) := 'NO NAME'; // AxisName is limited to 30 chars, IdxGrp := 4000 + _AxisRef.NcToPlc.AxisId, IdxOffs := 16#02
  stEncoderType               : STRING(30) := 'NO TYPE';
  eEncoderType                : E_AxisEncoderType;
  
  // Motion Control FB Instances
  fbPower                     : MC_Power;
  fbReset                     : MC_Reset;
  fbHalt                      : MC_Halt;
  fbStop                      : MC_Stop;
  fbHome                      : MC_Home;
  fbJog                       : MC_Jog;

  fbReadParameter             : MC_ReadParameter;
  fbWriteParameter            : Tc2_MC2.MC_WriteParameter;
  fbMoveVelocity1             : MC_MoveVelocity;
  fbMoveVelocity2             : MC_MoveVelocity;
  fbMoveAbsolute1             : MC_MoveAbsolute;
  fbMoveAbsolute2             : MC_MoveAbsolute;
  fbMoveEndless               : Tc2_MC2.MC_MoveContinuousAbsolute;

  // ADS read instance for reading startup information from NC
  fbADSRead                   : ADSREAD;

  // private vars for Methode Params
  stHaltParams                : ST_HaltParams;
  stHomeParams                : ST_HomeParams;
  stJogParams                 : ST_JogParams;
  stMoveAbsParams             : ST_MoveAbsParams;
  stMoveVeloParams            : ST_MoveVeloParams;
  stReadParamParams           : ST_ReadParamParams; 
  stStopParams                : ST_StopParams;
  stWriteParamParams          : ST_WriteParamParams;

  // local message list for online debug
  stMsg                       : ST_Message;
  atMsg                       : ARRAY[1..MAX_MSG_INTERN] OF ST_Message;
  itMsg                       : DINT := 1;

  // startup states for getting ADS information from NC
  _nStartUpErrorState,
  _nStartUp                   : DINT := 0;

  _bStartUpError,
  _bStartUp                   : BOOL;

  _uiEncoderType              : UDINT;

  _rCycleTime                 : LREAL;
  fbGetCurTaskIndex           : Tc2_System.GETCURTASKINDEX;

END_VAR
VAR CONSTANT
  MAX_MSG_INTERN              : DINT := 10;
END_VAR

fbPower(Axis:= _AxisRef);
_AxisRef();

IF NOT _bStartUp
THEN
  CASE _nStartUp OF
    0:
      // wait for cyclic data to be valid / connected
      IF (_AxisRef.NcToPlc.AxisId > 0)
      THEN
        fbADSRead(NETID       := '', 
                  PORT        := 501, 
                  IDXGRP      := (16#5000 + _AxisRef.NcToPlc.AxisId), 
                  IDXOFFS     := 16#00000003, // offset for encoder type
                  LEN         := SIZEOF(_uiEncoderType), 
                  DESTADDR    := ADR(_uiEncoderType),
                  TMOUT       := T#200MS,
                  READ        := FALSE);

        // clear required ADS information
        stAxisName            := 'NO NAME';
        _uiEncoderType        :=  0;
        _nStartUpErrorState   :=  0;  // debug
        _nStartUp             := 10;
      END_IF

  10:
    fbADSRead(NETID           := '', 
              PORT            := 501, 
              IDXGRP          := (16#5000 + _AxisRef.NcToPlc.AxisId), 
              IDXOFFS         := 16#00000003, // offset for encoder type
              LEN             := SIZEOF(_uiEncoderType), 
              DESTADDR        := ADR(_uiEncoderType),
              READ            := TRUE);

    IF fbADSRead.ERR
    THEN
      stMsg.eType             := E_MessageType.eMessageError;
      stMsg.eDevice           := e_Device.Axis;
      stMsg.eSubdevice        := e_Subdevice.General;
      stMsg.iErrorNumber      := fbAdsRead.ERRID;
      stMsg.sText             := 'StartUp Ads Error Read Encoder Type';

      MsgAdd(stMsg);
      f_MessageSet(stMsg);

      _nStartUpErrorState     := _nStartUp; // debug

      _nStartUp               := 90;

    ELSIF (_uiEncoderType > 0)
    THEN
      eEncoderType            := _uiEncoderType;
      stEncoderType           := TO_STRING(eEncoderType);

      fbADSRead(NETID         := '', 
                PORT          := 501, 
                IDXGRP        := (16#4000 + _AxisRef.NcToPlc.AxisId), 
                IDXOFFS       := 16#00000002, // offset for axis name
                LEN           := SIZEOF(stAxisName), 
                DESTADDR      := ADR(stAxisName),
                READ          := FALSE);

      _nStartUp               := 20;
    END_IF

  20:
    // the name must be read last, 
    // because this indicates the startup is done 
    // FB_AxisController is checking this entry
    fbADSRead(NETID           := '', 
              PORT            := 501, 
              IDXGRP          := (16#4000 + _AxisRef.NcToPlc.AxisId), 
              IDXOFFS         := 16#00000002, // offset for axis name
              LEN             := SIZEOF(stAxisName), 
              DESTADDR        := ADR(stAxisName),
              READ            := TRUE);
    IF fbADSRead.ERR
    THEN
      stMsg.eType             := E_MessageType.eMessageError;
      stMsg.eDevice           := e_Device.Axis;
      stMsg.eSubdevice        := e_Subdevice.General;
      stMsg.iErrorNumber      := fbAdsRead.ERRID;
      stMsg.sText             := 'StartUp Ads Error Read Axis Name';

      MsgAdd(stMsg);
      f_MessageSet(stMsg);

      _nStartUpErrorState     := _nStartUp; // debug

      _nStartUp               := 90;

    ELSIF (stAxisName <> 'NO NAME')
    THEN
      fbADSRead(READ          := FALSE);
      _nStartUp               := 100;
    END_IF

  90:
    _bStartUpError            := TRUE;
    _bStartUp                 := FALSE;

  100:
    _bStartUpError            := FALSE;
    _bStartUp                 := TRUE;
    _nStartUp                 := 0;
  END_CASE
END_IF

IF (_AxisRef.NcToPlc.AxisId > 0)
THEN
  ParamCheck();
END_IF

(* Write only; If plc cam is used for homing, this property needs to be set to the address of the calibration cam input prior to calling the Home methode *)
PROPERTY CalibrationCam : POINTER TO BOOL
SET
IF CalibrationCam <> 0 THEN
  pCalibrationCam := CalibrationCam;
END_IF
END_SET
END_PROPERTY

METHOD Clear : BOOL
VAR_INPUT
END_VAR
fbMoveAbsolute1 (Axis   := _AxisRef, Execute:= FALSE);
fbMoveAbsolute2 (Axis   := _AxisRef, Execute:= FALSE);
fbMoveEndless   (Axis   := _AxisRef, Execute:= FALSE);
fbMoveVelocity1 (Axis   := _AxisRef, Execute:= FALSE);
fbMoveVelocity2 (Axis   := _AxisRef, Execute:= FALSE);
fbStop          (Axis   := _AxisRef, Execute:= FALSE);
fbReset         (Axis   := _AxisRef, Execute:= FALSE);
fbHalt          (Axis   := _AxisRef, Execute:= FALSE);
END_METHOD

(* Axis will be enabled (=> Control Release will be set) or disabled (=> Control Release will be reseted) by this property. Refer to MC_Power Function Block in the Tc2_MC2 library *)
PROPERTY Enable : BOOL
GET
Enable := fbPower.Status;
END_GET
SET
fbPower.Enable := Enable;
END_SET
END_PROPERTY

PROPERTY EncoderType : E_AxisEncoderType
GET
EncoderType := eEncoderType;
END_GET
END_PROPERTY

{attribute '''NORMAL__COMMENT' := ' Will try to reset an active error; Refer to MC_Reset Function Block in the Tc2_MC2 library '}
(* Will try to reset an active error; Refer to MC_Reset Function Block in the Tc2_MC2 library *)
METHOD ErrorReset : Tc2_MC2.ST_McOutputs
VAR_INPUT
  Execute : BOOL;
END_VAR
VAR_INST
  res    : Tc2_MC2.ST_McOutputs;
  nState : DINT;
END_VAR
CASE nState OF
  0:
    IF Execute
    THEN
      memset(ADR(res),0,SIZEOF(res));
      res.Busy                := TRUE;

      fbReset(Axis            := _AxisRef,
              Execute         := FALSE);

      nState                  := 10;
    END_IF
END_CASE
CASE nState OF
  10:
    fbReset(Axis              := _AxisRef,
            Execute           := TRUE);

    IF fbReset.Done
    THEN
      fbReset(Axis            := _AxisRef,
              Execute         := FALSE);

      _nStartUp               := 0;
      nState                  := 20;
    ELSE
      IF fbReset.Error
      THEN
        res.ErrorID           := fbReset.ErrorID;

        stMsg.eType           := E_MessageType.eMessageError;
        stMsg.eDevice         := e_Device.Axis + TO_DINT(_AxisRef.NcToPlc.AxisId);
        stMsg.eSubdevice      := e_SubDevice.fbReset;
        stMsg.iErrorNumber    := fbReset.ErrorID;

        f_MessageSet(stMsg);
        MsgAdd(stMsg);

        fbReset(Axis          := _AxisRef,
                Execute       := FALSE);

        nState                := 99;
      ELSIF NOT fbReset.Busy
      THEN
        fbReset(Axis          := _AxisRef,
                Execute       := FALSE);
  
        nState                := 20;
      END_IF
    END_IF
END_CASE
CASE nState OF
  20:
    res.Busy                  := FALSE;
    res.Done                  := TRUE;
  
  99:
    res.Busy                  := FALSE;
    res.Error                 := TRUE;
END_CASE

IF NOT Execute
THEN
  memset(ADR(res),0,SIZEOF(res));
  nState                      := 0;
END_IF

ErrorReset := res;
END_METHOD

(* Enables Movement in negative direction if set to TRUE. Refer to MC_Power Function Block in the Tc2_MC2 library *)
PROPERTY FeedEnable_Negative : BOOL
GET
FeedEnable_Negative := fbPower.Enable_Negative;
END_GET
SET
fbPower.Enable_Negative := FeedEnable_Negative;
END_SET
END_PROPERTY

(* Enables Movement in positive direction if set to TRUE. Refer to MC_Power Function Block in the Tc2_MC2 library *)
PROPERTY FeedEnable_Positive : BOOL
GET
FeedEnable_Positive := fbPower.Enable_Positive;
END_GET
SET
fbPower.Enable_Positive := FeedEnable_Positive;
END_SET
END_PROPERTY

{attribute '''NORMAL__COMMENT' := ' Halt stops an axis with a defined braking ramp. In contrast to Stop, the axis is not locked against further movement commands. The axis can therefore
  be restarted through a further command during the braking ramp or after it has come to a halt. Refer to MC_Halt Function Block in the Tc2_MC2 library '}
(* Halt stops an axis with a defined braking ramp. In contrast to Stop, the axis is not locked against further movement commands. The axis can therefore
  be restarted through a further command during the braking ramp or after it has come to a halt. Refer to MC_Halt Function Block in the Tc2_MC2 library *)
METHOD Halt : Tc2_MC2.ST_McOutputs
VAR_INPUT
  Execute : BOOL;
  (* Deceleration. If not specified, DefaultDeceleration will be used. For safety reasons MC_Halt and MC_Stop cannot be executed 
                with weaker dynamics than the currently active travel command. The parameterization is adjusted automatically, if necessary *)
  {attribute '''NORMAL__COMMENT' := ' Deceleration. If not specified, DefaultDeceleration will be used. For safety reasons MC_Halt and MC_Stop cannot be executed 
                with weaker dynamics than the currently active travel command. The parameterization is adjusted automatically, if necessary '}
  Deceleration  : LREAL;
  (* Jerk. If not specified, DefaultJerk will be used. For safety reasons MC_Halt and MC_Stop cannot be executed 
                with weaker dynamics than the currently active travel command. The parameterization is adjusted automatically, if necessary *)
  {attribute '''NORMAL__COMMENT' := ' Jerk. If not specified, DefaultJerk will be used. For safety reasons MC_Halt and MC_Stop cannot be executed 
                with weaker dynamics than the currently active travel command. The parameterization is adjusted automatically, if necessary '}
  Jerk  : LREAL;
  (* The BufferMode is analyzed, if the axis is already executing another command. The running command can be aborted,
                    or the new command becomes active after the running command. The BufferMode also determines the transition condition from 
                    the current to the next command. If the command is applied to a coupled slave axis used, the only available buffer mode is Aborting.
                    Special characteristics of MC_Halt: The MC_buffer mode has no effect, if the command is executed when the system is at a standstill.
                    The blending modes MC_BlendingNext andMC_BlendingLow do not change the last target position, although they can result in a change in
                    dynamics (deceleration) of the stop ramp. The modes MC_BlendingPrevious andMC_BlendingHigh extend the travel to the original target position.
                    The stop ramp is only initiated when this position is reached (defined braking point). *)
  {attribute '''NORMAL__COMMENT' := ' The BufferMode is analyzed, if the axis is already executing another command. The running command can be aborted,
                    or the new command becomes active after the running command. The BufferMode also determines the transition condition from 
                    the current to the next command. If the command is applied to a coupled slave axis used, the only available buffer mode is Aborting.
                    Special characteristics of MC_Halt: The MC_buffer mode has no effect, if the command is executed when the system is at a standstill.
                    The blending modes MC_BlendingNext andMC_BlendingLow do not change the last target position, although they can result in a change in
                    dynamics (deceleration) of the stop ramp. The modes MC_BlendingPrevious andMC_BlendingHigh extend the travel to the original target position.
                    The stop ramp is only initiated when this position is reached (defined braking point). '}
  BufferMode  : Tc2_MC2.MC_BufferMode;
END_VAR
VAR_INST
  res       : Tc2_MC2.ST_McOutputs;
  nState    : DINT;
  fUsedDec,
  fUsedJerk : LREAL;
  itmp      : ARRAY[1..3] OF DINT;
END_VAR
IF NOT Execute
THEN
  memset(ADR(res),0,SIZEOF(res));
  nState                    := 0;
END_IF


CASE nState OF
  0:
    IF Execute
    THEN
      memset(ADR(res),  0, SIZEOF(res));
      memset(ADR(itmp), 0, SIZEOF(itmp));

      res.Busy              := TRUE;

      fUsedDec := SEL((Deceleration = 0),Deceleration, stDefaultDeceleration.fValue);
      fUsedJerk:= SEL((Jerk = 0),Jerk, stDefaultJerk.fValue);

      fbHalt(Axis           := _AxisRef, 
             Execute        := FALSE, 
             Deceleration   := fUsedDec, 
             Jerk           := fUsedJerk, 
             BufferMode     := Tc2_MC2.MC_BufferMode.MC_Aborting);

      nState := 10;
    END_IF
END_CASE
CASE nState OF
  10:
    fbHalt(Axis             := _AxisRef, 
           Execute          := TRUE);

    IF _AxisRef.Status.Stopping
    THEN
      nState                := 30;
    ELSE
      itmp[1]               := itmp[1] + 1;

      IF (itmp[1] MOD 100 = 0)
      THEN
        fbHalt(Axis         := _AxisRef, 
               Execute      := FALSE);

        fbStop(Axis         := _AxisRef, 
               Execute      := TRUE);

        stMsg.eType         := E_MessageType.eMessageInfo;
        stMsg.eDevice       := e_Device.Axis + TO_DINT(_AxisRef.NcToPlc.AxisId);
        stMsg.eSubdevice    := e_SubDevice.fbHalt;
        stMsg.iErrorNumber  := _AxisRef.NcToPlc.AxisId;
        stMsg.sText         := 'timeout 1 stopping';
        f_MessageSet(stMsg);

        nState              := 15;
      END_IF
    END_IF

    IF fbHalt.Error
    THEN
      res.ErrorID           := fbHalt.ErrorID;
      stMsg.eType           := E_MessageType.eMessageError;
      stMsg.eDevice         := e_Device.Axis + TO_DINT(_AxisRef.NcToPlc.AxisId);
      stMsg.eSubdevice      :=  e_SubDevice.fbHalt;
      stMsg.iErrorNumber    := fbHalt.ErrorID;

      f_MessageSet(stMsg);
      MsgAdd(stMsg);

      nState                := 99;
    END_IF
END_CASE
CASE nState OF
  15:
    fbStop(Axis             := _AxisRef, 
           Execute          := TRUE);

    IF _AxisRef.Status.Stopping
    THEN
      nState                := 30;
    ELSE
      itmp[2]               := itmp[2] + 1;

      IF (itmp[2] MOD 50 = 0)
      THEN
        fbStop (Axis        := _AxisRef, 
                Execute     := FALSE);

        fbReset(Axis        := _AxisRef, 
                Execute     := TRUE);

        stMsg.eType         := E_MessageType.eMessageInfo;
        stMsg.eDevice       := e_Device.Axis + TO_DINT(_AxisRef.NcToPlc.AxisId);
        stMsg.eSubdevice    := e_SubDevice.fbStop;
        stMsg.iErrorNumber  := _AxisRef.NcToPlc.AxisId;
        stMsg.sText         := 'timeout 2 reset';

        f_MessageSet(stMsg);

        nState              := 20;
      END_IF
    END_IF
END_CASE
CASE nState OF
  20:
    IF _AxisRef.Status.NotMoving
    THEN
      fbReset(Axis          := _AxisRef, 
              Execute       := FALSE);

      nState                := 40;
    ELSE
      itmp[3]               := itmp[3] + 1;

      IF (itmp[3] MOD 100 = 0)
      THEN
        fbStop (Axis        := _AxisRef, 
                Execute     := FALSE);

        fbReset(Axis        := _AxisRef, 
                Execute     := FALSE);

        stMsg.eType         := E_MessageType.eMessageInfo;
        stMsg.eDevice       := e_Device.Axis + TO_DINT(_AxisRef.NcToPlc.AxisId);
        stMsg.eSubdevice    := e_SubDevice.fbReset;
        stMsg.iErrorNumber  := _AxisRef.NcToPlc.AxisId;
        stMsg.sText         := 'timeout 3 retry';

        f_MessageSet(stMsg);

        nState              := 15;
      END_IF
    END_IF
END_CASE
CASE nState OF
  30:
    IF _AxisRef.Status.NotMoving
    THEN
      fbStop(Axis           := _AxisRef, 
             Execute        := FALSE);

      fbReset(Axis          := _AxisRef, 
              Execute       := TRUE);

      nState                := 39;
    END_IF
END_CASE
CASE nState OF
  39:
    fbReset(Axis            := _AxisRef, 
            Execute         := FALSE);

    nState                  := 40;
END_CASE
CASE nState OF
  40:
    res.Error               := FALSE;
    res.Busy                := FALSE;
    res.Done                := TRUE;

  99:
    res.Error               := TRUE;
    res.Busy                := FALSE;
    res.Done                := FALSE;
END_CASE



Halt := res;
END_METHOD

{attribute '''NORMAL__COMMENT' := ' Initiates the calibration of the coordinates of the NC axis referencing). Certain parameters of the NC axis will have influence on the behavior
  Will return without action if HomingMode equals MC_DefaultHoming and CalibrationCam property is not set; in case of MC_DefaultHoming the property 
  CalibrationCam has to be set prior to calling this methode. Refer to MC_Home Function Block in the Tc2_MC2 library '}
(* Initiates the calibration of the coordinates of the NC axis referencing). Certain parameters of the NC axis will have influence on the behavior
  Will return without action if HomingMode equals MC_DefaultHoming and CalibrationCam property is not set; in case of MC_DefaultHoming the property 
  CalibrationCam has to be set prior to calling this methode. Refer to MC_Home Function Block in the Tc2_MC2 library *)
METHOD Home : Tc2_MC2.ST_McOutputs
VAR_INPUT
  Execute   : BOOL;
  (* Absolute reference position to which the axis is set after homing.
                          The Default setting DEFAULT_HOME_POSITION, the Reference position for homing specified in the TwinCAT System Manager is used.
                          Attention: Since the reference position is generally set during the motion, the axis will not stop exactly at this position. 
                          The standstill position differs by the braking distance of the axis, although the calibration is nevertheless exact *)
  {attribute '''NORMAL__COMMENT' := ' Absolute reference position to which the axis is set after homing.
                          The Default setting DEFAULT_HOME_POSITION, the Reference position for homing specified in the TwinCAT System Manager is used.
                          Attention: Since the reference position is generally set during the motion, the axis will not stop exactly at this position. 
                          The standstill position differs by the braking distance of the axis, although the calibration is nevertheless exact '}
  Position  : LREAL := DEFAULT_HOME_POSITION;
  (* determines in which way the calibration is carried out: 
                                MC_DefaultHoming initiates standard homing; 
                                MC_Direct sets the axis position directly to Position without executing a movement.
                                MC_ForceCalibration enforces the "axis is calibrated" state. No movement takes place, and the position remains unchanged; 
                                MC_ResetCalibration resets the calibration state of the axis. No movement takes place, and the position remains unchanged. *)
  {attribute '''NORMAL__COMMENT' := ' determines in which way the calibration is carried out: 
                                MC_DefaultHoming initiates standard homing; 
                                MC_Direct sets the axis position directly to Position without executing a movement.
                                MC_ForceCalibration enforces the "axis is calibrated" state. No movement takes place, and the position remains unchanged; 
                                MC_ResetCalibration resets the calibration state of the axis. No movement takes place, and the position remains unchanged. '}
  HomingMode  : Tc2_MC2.MC_HomingMode := MC_DefaultHoming;
  (* Options.ClearPositionLag is only active in mode MC_Direct and can optionally be used to set the set and actual positions to the same value.
                      In this case the following error is cancelled. *)
  {attribute '''NORMAL__COMMENT' := ' Options.ClearPositionLag is only active in mode MC_Direct and can optionally be used to set the set and actual positions to the same value.
                      In this case the following error is cancelled. '}
  Options : Tc2_MC2.ST_HomingOptions;
END_VAR
VAR_INST
  res       : Tc2_MC2.ST_McOutputs;
  nState    : DINT;
  fUsedDec,
  fUsedJerk : LREAL;
END_VAR
// do nothing if at Default Homing Mode Property CalibrationCam is invalid
IF (HomingMode = MC_DefaultHoming) 
THEN
  IF (pCalibrationCam = 0) 
  THEN
    res.Error                 := TRUE;
    res.ErrorID               := 666;
    Home                      := res;
    RETURN;
  ELSE 
    fbHome.bCalibrationCam    := pCalibrationCam^;
  END_IF
END_IF


CASE nState OF
  0:
    IF Execute
    THEN
      memset(ADR(res),0,SIZEOF(res));
      res.Busy                := TRUE;

      fbHome(Axis             := _AxisRef, 
             Execute          := FALSE, 
             Position         := Position, 
             HomingMode       := HomingMode, 
             BufferMode       := , 
             Options          := Options, 
             bCalibrationCam  := pCalibrationCam^);

      nState                  := 10;
    END_IF
END_CASE
CASE nState OF
  10:
    fbHome(Execute            := TRUE, 
           Axis               := _AxisRef);

    IF fbHome.Done
    THEN
      fbHome(Execute          := FALSE, 
             Axis             := _AxisRef);

      nState                  := 20;

    ELSE
      IF fbHome.Error
      THEN
        res.ErrorID           := fbHome.ErrorID;

        stMsg.eType           := E_MessageType.eMessageError;
        stMsg.eDevice         := e_Device.Axis + TO_DINT(_AxisRef.NcToPlc.AxisId);
        stMsg.eSubdevice      :=  e_SubDevice.fbHome;
        stMsg.iErrorNumber    := fbHome.ErrorID;

        f_MessageSet(stMsg);
        MsgAdd(stMsg);

        fbHome(Execute        := FALSE, 
               Axis           := _AxisRef);

        nState                := 99;
      END_IF
    END_IF
END_CASE
CASE nState OF
  20:
    res.Error                 := FALSE;
    res.Busy                  := FALSE;
    res.Done                  := TRUE;

END_CASE
CASE nState OF
  99:
    res.Error                 := TRUE;
    res.Busy                  := FALSE;
    res.Done                  := FALSE;
END_CASE

IF NOT Execute
THEN
  memset(ADR(res),0,SIZEOF(res));
  nState                      := 0;
END_IF

Home := res;
END_METHOD

{attribute '''NORMAL__COMMENT' := ' This methode provides easy to use manual motion commands by the JogForward and JogBackwards inputs. The required operating mode is specified via the mode input. 
  An inching mode for moving the axis by a specified distance whenever the JogForward and JogBackwards inputs are set is  also available. The velocity and dynamics 
  of the motion can be specified depending on the mode. If the mode is not an inching mode, the methode needs to be called cyclically for proper evaluation of the Jog Inputs.
  Refer to MC_JOG Function Block in the Tc2_MC2 library '}
(* This methode provides easy to use manual motion commands by the JogForward and JogBackwards inputs. The required operating mode is specified via the mode input. 
  An inching mode for moving the axis by a specified distance whenever the JogForward and JogBackwards inputs are set is  also available. The velocity and dynamics 
  of the motion can be specified depending on the mode. If the mode is not an inching mode, the methode needs to be called cyclically for proper evaluation of the Jog Inputs.
  Refer to MC_JOG Function Block in the Tc2_MC2 library *)
METHOD Jog : Tc2_MC2.ST_McOutputs
VAR_INPUT
  (* The command is executed with increasing edge, and the axis is moved in positive direction of travel. Depending on the mode, the axis moves as long as 
              the signal remains TRUE, or it stops automatically after a specified distance. During the motion no further signal edges are accepted 
              (this includes the JogBackwards input). If signal edges occur simultaneously at the JogForward and JogBackwards inputs, JogForward has priority *)
  {attribute '''NORMAL__COMMENT' := ' The command is executed with increasing edge, and the axis is moved in positive direction of travel. Depending on the mode, the axis moves as long as 
              the signal remains TRUE, or it stops automatically after a specified distance. During the motion no further signal edges are accepted 
              (this includes the JogBackwards input). If signal edges occur simultaneously at the JogForward and JogBackwards inputs, JogForward has priority '}
  JogForward  : BOOL;
  (* The command is executed with increasing edge, and the axis is moved in negative direction of travel. JogForward and JogBackwards should be triggered 
              alternatively, although they are also mutually locked internally *)
  {attribute '''NORMAL__COMMENT' := ' The command is executed with increasing edge, and the axis is moved in negative direction of travel. JogForward and JogBackwards should be triggered 
              alternatively, although they are also mutually locked internally '}
  JogBackwards  : BOOL;
  (* The Mode input determines the operating mode in which the manual function is executed.
          MC_JOGMODE_STANDARD_SLOW The axis is moved as long as the signal at one of the jog inputs is TRUE. The low velocity for manual functions specified in the TwinCAT 
            System Manager and standard dynamics are used. In this mode the position, velocity and dynamics data specified in the function block have no effect. 
          MC_JOGMODE_STANDARD_FAST.The axis is moved as long as the signal at one of the jog inputs is TRUE. The high velocity for manual functions specified in the TwinCAT
            System Manager and standard dynamics are used. In this mode the position, velocity and dynamics data specified in the function block have no effect. 
          MC_JOGMODE_CONTINOUS The axis is moved as long as the signal at one of the jog inputs is TRUE. The velocity and dynamics data specified by the user are used.
            The position has no effect.
          MC_JOGMODE_INCHING.With rising edge at one of the jog inputs the axis is moved by a certain distance, which is specified via the position input. The axis stops
            automatically, irrespective of the state of the jog inputs. A new movement step is only executed once a further rising edge is encountered. At each start 
            the velocity and dynamics data specified by the user are used. 
          MC_JOGMODE_INCHING_MODULO.With rising edge at one of the jog inputs the axis is moved by a certain distance, which is specified via the position input. The axis
            position will snap to an integer multiple of the position parameter. The axis stops automatically, irrespective of the state of the jog inputs. A new movement
            step is only executed once a further rising edge is encountered. With each start the velocity and dynamics data specified by the user are used *)
  {attribute '''NORMAL__COMMENT' := ' The Mode input determines the operating mode in which the manual function is executed.
          MC_JOGMODE_STANDARD_SLOW The axis is moved as long as the signal at one of the jog inputs is TRUE. The low velocity for manual functions specified in the TwinCAT 
            System Manager and standard dynamics are used. In this mode the position, velocity and dynamics data specified in the function block have no effect. 
          MC_JOGMODE_STANDARD_FAST.The axis is moved as long as the signal at one of the jog inputs is TRUE. The high velocity for manual functions specified in the TwinCAT
            System Manager and standard dynamics are used. In this mode the position, velocity and dynamics data specified in the function block have no effect. 
          MC_JOGMODE_CONTINOUS The axis is moved as long as the signal at one of the jog inputs is TRUE. The velocity and dynamics data specified by the user are used.
            The position has no effect.
          MC_JOGMODE_INCHING.With rising edge at one of the jog inputs the axis is moved by a certain distance, which is specified via the position input. The axis stops
            automatically, irrespective of the state of the jog inputs. A new movement step is only executed once a further rising edge is encountered. At each start 
            the velocity and dynamics data specified by the user are used. 
          MC_JOGMODE_INCHING_MODULO.With rising edge at one of the jog inputs the axis is moved by a certain distance, which is specified via the position input. The axis
            position will snap to an integer multiple of the position parameter. The axis stops automatically, irrespective of the state of the jog inputs. A new movement
            step is only executed once a further rising edge is encountered. With each start the velocity and dynamics data specified by the user are used '}
  Mode  : Tc2_MC2.E_JogMode;
  (* Relative distance for movements in MC_JOGMODE_INCHING mode *)
  {attribute '''NORMAL__COMMENT' := ' Relative distance for movements in MC_JOGMODE_INCHING mode '}
  Position  : LREAL;
  (* Maximum travel velocity. If not specified, DefaultVelocity will be used *)
  {attribute '''NORMAL__COMMENT' := ' Maximum travel velocity. If not specified, DefaultVelocity will be used '}
  Velocity  : LREAL;
  (* Acceleration. If not specified, DefaultAcceleration will be used *)
  {attribute '''NORMAL__COMMENT' := ' Acceleration. If not specified, DefaultAcceleration will be used '}
  Acceleration  : LREAL;
  (* Deceleration. If not specified, DefaultDeceleration will be used *)
  {attribute '''NORMAL__COMMENT' := ' Deceleration. If not specified, DefaultDeceleration will be used '}
  Deceleration  : LREAL;
  (* Jerk. If not specified, DefaultJerk will be used *)
  {attribute '''NORMAL__COMMENT' := ' Jerk. If not specified, DefaultJerk will be used '}
  Jerk  : LREAL;
END_VAR
VAR_INST
  rtrigErr  : Tc2_Standard.R_TRIG;
  fUsedVel, 
  fUsedAcc, 
  fUsedDec, 
  fUsedJrk  : LREAL;
END_VAR
// Select Default values of dynamic parameter if 0 is specified
fUsedVel := SEL((Velocity = 0),     Velocity,     fDefaultVelocity);
fUsedAcc := SEL((Acceleration = 0), Acceleration, stDefaultAcceleration.fValue);
fUsedDec := SEL((Deceleration = 0), Deceleration, stDefaultDeceleration.fValue);
fUsedJrk := SEL((Jerk = 0),         Jerk,         stDefaultJerk.fValue);


// call fbJog
fbJog(Axis                  := _AxisRef, 
      JogForward            := JogForward, 
      JogBackwards          := JogBackwards, 
      Mode                  := Mode, 
      Position              := Position, 
      Velocity              := fUsedVel, 
      Acceleration          := fUsedAcc, 
      Deceleration          := fUsedDec, 
      Jerk                  := fUsedJrk);


rtrigErr(CLK                := fbJog.Error);


stJogParams.Acceleration    := Acceleration;
stJogParams.Deceleration    := Deceleration;
stJogParams.Jerk            := Jerk;
stJogParams.JogBackwards    := JogBackwards;
stJogParams.JogForward      := JogForward;
stJogParams.Mode            := Mode;
stJogParams.Position        := Position;
stJogParams.Velocity        := Velocity;

// return status
Jog.Active                  := fbJog.Active;
Jog.Busy                    := fbJog.Busy;
Jog.CommandAborted          := fbJog.CommandAborted;
Jog.Done                    := fbJog.Done;
Jog.Error                   := fbJog.Error;
Jog.ErrorID                 := fbJog.ErrorID;

// push error
IF rtrigErr.Q
THEN
  // write list entry
  stMsg.eType               := E_MessageType.eMessageError;
  stMsg.eDevice             := e_Device.Axis + TO_DINT(_AxisRef.NcToPlc.AxisId);
  stMsg.eSubdevice          :=  e_SubDevice.fbJog;
  stMsg.iErrorNumber        := fbJog.ErrorID;

  f_MessageSet(stMsg);
  MsgAdd(stMsg);
END_IF
END_METHOD

METHOD LocalParameterReload : BOOL
VAR_INPUT
END_VAR

stSwPosLimitNegativeActive.bValid   := FALSE;
stSwPosLimitPositiveActive.bValid   := FALSE;

stDefaultAcceleration.bValid        := FALSE;
stDefaultDeceleration.bValid        := FALSE;

stDefaultJerk.bValid                := FALSE;

stMaxAcceleration.bValid            := FALSE;
stMaxDeceleration.bValid            := FALSE;

stMaxVelocity.bValid                := FALSE;

stSwPosLimitNegative.bValid         := FALSE;
stSwPosLimitPositive.bValid         := FALSE;

stHomingSearchVelo.bValid           := FALSE;

stHomingVelo.bValid                 := FALSE;

stTargetPositionWindow.bValid       := FALSE;

LocalParameterReload                := TRUE;
END_METHOD

{attribute '''NORMAL__COMMENT' := ' MoveAbsolute starts positioning to an absolute target position with monitoring of the axis movement over the whole travel path. Refer to MC_MoveAbsolute Function Block in the
  Tc2_MC2 library. To instances of MC_MoveAbsolute are used to trigger new parameter during movement; Use Buffermode to control the transition. '}
(* MoveAbsolute starts positioning to an absolute target position with monitoring of the axis movement over the whole travel path. Refer to MC_MoveAbsolute Function Block in the
  Tc2_MC2 library. To instances of MC_MoveAbsolute are used to trigger new parameter during movement; Use Buffermode to control the transition. *)
METHOD MoveAbsolute : Tc2_MC2.ST_McOutputs
VAR_INPUT
  Enable    : BOOL;
  (* Absolute target position to be used for positioning *)
  {attribute '''NORMAL__COMMENT' := ' Absolute target position to be used for positioning '}
  Position  : LREAL;
  (* Maximum travel velocity. If not specified, DefaultVelocity will be used *)
  {attribute '''NORMAL__COMMENT' := ' Maximum travel velocity. If not specified, DefaultVelocity will be used '}
  Velocity  : LREAL;
  (* Acceleration. If not specified, DefaultAcceleration will be used *)
  {attribute '''NORMAL__COMMENT' := ' Acceleration. If not specified, DefaultAcceleration will be used '}
  Acceleration  : LREAL;
  (* Deceleration. If not specified, DefaultDeceleration will be used *)
  {attribute '''NORMAL__COMMENT' := ' Deceleration. If not specified, DefaultDeceleration will be used '}
  Deceleration  : LREAL;
  (* Jerk. If not specified, DefaultJerk will be used *)
  {attribute '''NORMAL__COMMENT' := ' Jerk. If not specified, DefaultJerk will be used '}
  Jerk  : LREAL;
  (* The BufferMode is analyzed, if the axis is already executing another command. The running command can be aborted,
                    or the new command becomes active after the running command. The BufferMode also determines the transition condition from the current to the next command.
                    If the command is applied to a coupled slave axis used, the only available buffer mode is Aborting. *)
  {attribute '''NORMAL__COMMENT' := ' The BufferMode is analyzed, if the axis is already executing another command. The running command can be aborted,
                    or the new command becomes active after the running command. The BufferMode also determines the transition condition from the current to the next command.
                    If the command is applied to a coupled slave axis used, the only available buffer mode is Aborting. '}
  BufferMode  : Tc2_MC2.MC_BufferMode;
END_VAR
VAR_IN_OUT
  fActivePosition   : LREAL;
  eState            : e_AxisFunction;
END_VAR
VAR_INST
  bLog      : BOOL;
  res       : Tc2_MC2.ST_McOutputs;
  nState    : DINT;
  fUsedPos,
  fUsedVel,
  fUsedAcc,
  fUsedDec,
  fUsedJrk    : LREAL;
END_VAR
// Select Default values of dynamic parameter if 0 is specified
fUsedVel := Velocity;
fUsedAcc := Acceleration;
fUsedDec := Deceleration;
fUsedJrk := Jerk;


CASE nState OF
  0:
    IF Enable
    THEN
      memset(ADR(res),0,SIZEOF(res));
      res.Busy                      := TRUE;
      fUsedPos                      := Position;

      fbMoveAbsolute1(Axis          := _AxisRef, 
                      Execute       := FALSE);

      fbMoveAbsolute2(Axis          := _AxisRef, 
                      Execute       := FALSE);

      nState                        := 10;

        stMsg.eType                 := E_MessageType.eMessageInfo;
        stMsg.eDevice               := e_Device.Axis + TO_DINT(_AxisRef.NcToPlc.AxisId);
        stMsg.eSubdevice            :=  e_SubDevice.fbMoveAbsolute1;
        stMsg.iErrorNumber          := nState;
        stMsg.sText                 := concat('MoveBuffer start: ', TO_STRING(fUsedPos));
        f_MessageSet(stMsg);
        MsgAdd(stMsg);
    END_IF
END_CASE
CASE nState OF
  10:
    eState                          := e_AxisFunction.AXIS_BUSY;
    fbMoveAbsolute1(Axis            := _AxisRef, 
                    Execute         := TRUE, 
                    Position        := fUsedPos,
                    Velocity        := fUsedVel, 
                    Acceleration    := fUsedAcc, 
                    Deceleration    := fUsedDec, 
                    Jerk            := fUsedJrk, 
                    BufferMode      := BufferMode);

      fbMoveAbsolute2(Axis          := _AxisRef, 
                      Execute       := FALSE);

    IF fbMoveAbsolute1.Error
    THEN
      stMsg.eType                 := E_MessageType.eMessageError;
      stMsg.eDevice               := e_Device.Axis + TO_DINT(_AxisRef.NcToPlc.AxisId);
      stMsg.eSubdevice            :=  e_SubDevice.fbMoveAbsolute1;
      stMsg.iErrorNumber          := fbMoveAbsolute1.ErrorID;
      f_MessageSet(stMsg);
      MsgAdd(stMsg);

      res.ErrorID                 := fbMoveAbsolute1.ErrorID;

      nState                      := 99;

    ELSIF fbMoveAbsolute1.Busy OR 
          fbMoveAbsolute1.Done
    THEN
      IF fbMoveAbsolute1.Active
      THEN
        nState                      := 20;
        stMsg.eType                 := E_MessageType.eMessageInfo;
        stMsg.eDevice               := e_Device.Axis + TO_DINT(_AxisRef.NcToPlc.AxisId);
        stMsg.eSubdevice            :=  e_SubDevice.fbMoveAbsolute1;
        stMsg.iErrorNumber          := nState;
        stMsg.sText                 := concat('MoveBuffer work: ', TO_STRING(fUsedPos));
        f_MessageSet(stMsg);
        MsgAdd(stMsg);
      END_IF
    END_IF
END_CASE
CASE nState OF
  20:
    fbMoveAbsolute1(Axis            := _AxisRef);

    fbMoveAbsolute2(Axis            := _AxisRef, 
                      Execute       := FALSE);

    res.Active                      := TRUE;

    IF fbMoveAbsolute1.Error
    THEN
      stMsg.eType                   := E_MessageType.eMessageError;
      stMsg.eDevice                 := e_Device.Axis + TO_DINT(_AxisRef.NcToPlc.AxisId);
      stMsg.eSubdevice              :=  e_SubDevice.fbMoveAbsolute1;
      stMsg.iErrorNumber            := fbMoveAbsolute1.ErrorID;
      f_MessageSet(stMsg);
      MsgAdd(stMsg);

      res.ErrorID                   := fbMoveAbsolute1.ErrorID;

      nState                        := 99;

    ELSIF (Position <> fUsedPos)
    THEN
      fbMoveAbsolute1(Axis          := _AxisRef, 
                    Execute         := FALSE); 

      nState                        := 30;

      stMsg.eType                   := E_MessageType.eMessageInfo;
      stMsg.eDevice                 := e_Device.Axis + TO_DINT(_AxisRef.NcToPlc.AxisId);
      stMsg.eSubdevice              :=  e_SubDevice.fbMoveAbsolute2;
      stMsg.iErrorNumber            := nState;
      stMsg.sText                   := concat('Pos changed: ', TO_STRING(fUsedPos));
      stMsg.sText                   := concat(stMsg.sText, ' to ');
      stMsg.sText                   := concat(stMsg.sText, TO_STRING(Position));

      f_MessageSet(stMsg);
      MsgAdd(stMsg);

      fUsedPos                      := Position;
    END_IF
END_CASE
CASE nState OF
  30:
    eState                          := e_AxisFunction.AXIS_ACK;
    fbMoveAbsolute2(  Axis          := _AxisRef, 
                      Execute       := TRUE,
                      Position      := fUsedPos, 
                      Velocity      := fUsedVel, 
                      Acceleration  := fUsedAcc, 
                      Deceleration  := fUsedDec, 
                      Jerk          := fUsedJrk, 
                      BufferMode    := BufferMode);

      fbMoveAbsolute1(Axis          := _AxisRef, 
                      Execute       := FALSE);

    IF fbMoveAbsolute2.Error
    THEN
      stMsg.eType                 := E_MessageType.eMessageError;
      stMsg.eDevice               := e_Device.Axis + TO_DINT(_AxisRef.NcToPlc.AxisId);
      stMsg.eSubdevice            :=  e_SubDevice.fbMoveAbsolute2;
      stMsg.iErrorNumber          := fbMoveAbsolute2.ErrorID;
      stMsg.sText                 := '';
      f_MessageSet(stMsg);
      MsgAdd(stMsg);

      res.ErrorID                 := fbMoveAbsolute2.ErrorID;

      nState                      := 99;


    ELSIF fbMoveAbsolute2.Busy OR
          fbMoveAbsolute2.Done
    THEN
      IF fbMoveAbsolute2.Active
      THEN
        nState                      := 40;
        stMsg.eType                 := E_MessageType.eMessageInfo;
        stMsg.eDevice               := e_Device.Axis + TO_DINT(_AxisRef.NcToPlc.AxisId);
        stMsg.eSubdevice            :=  e_SubDevice.fbMoveAbsolute2;
        stMsg.iErrorNumber          := nState;
        stMsg.sText                 := concat('MoveBuffer work: ', TO_STRING(fUsedPos));
        f_MessageSet(stMsg);
        MsgAdd(stMsg);
      END_IF
    END_IF
END_CASE
CASE nState OF
  40:
    fbMoveAbsolute1(Axis            := _AxisRef, 
                    Execute         := FALSE);

    fbMoveAbsolute2(Axis            := _AxisRef);

    res.Active                      := TRUE;

    IF fbMoveAbsolute2.Error
    THEN
      stMsg.eType                   := E_MessageType.eMessageError;
      stMsg.eDevice                 := e_Device.Axis + TO_DINT(_AxisRef.NcToPlc.AxisId);
      stMsg.eSubdevice              :=  e_SubDevice.fbMoveAbsolute2;
      stMsg.iErrorNumber            := fbMoveAbsolute2.ErrorID;
      stMsg.sText                   := '';
      f_MessageSet(stMsg);
      MsgAdd(stMsg);

      res.ErrorID                   := fbMoveAbsolute2.ErrorID;

      nState                        := 99;

    ELSIF (Position <> fUsedPos)
    THEN
      fbMoveAbsolute2(Axis          := _AxisRef, 
                      Execute       := FALSE);

      nState                        := 10;

      stMsg.eType                   := E_MessageType.eMessageInfo;
      stMsg.eDevice                 := e_Device.Axis + TO_DINT(_AxisRef.NcToPlc.AxisId);
      stMsg.eSubdevice              :=  e_SubDevice.fbMoveAbsolute1;
      stMsg.iErrorNumber            := nState;
      stMsg.sText                   := concat('Pos changed: ', TO_STRING(fUsedPos));
      stMsg.sText                   := concat(stMsg.sText, ' to ');
      stMsg.sText                   := concat(stMsg.sText, TO_STRING(Position));
      f_MessageSet(stMsg);
      MsgAdd(stMsg);

      fUsedPos                      := Position;
    END_IF
END_CASE
CASE nState OF
  99:
    res.Busy                        := FALSE;
    res.Error                       := TRUE;
    fbMoveAbsolute1(Axis            := _AxisRef, 
                    Execute         := FALSE);
  
    fbMoveAbsolute2(Axis            := _AxisRef, 
                    Execute         := FALSE);
END_CASE

IF NOT Enable
THEN
  eState                        := e_AxisFunction.AXIS_DISABLE;
  fUsedPos                      := 0.0;
  memset(ADR(res),0,SIZEOF(res));

  fbMoveAbsolute1(Axis          := _AxisRef, 
                  Execute       := FALSE);

  fbMoveAbsolute2(Axis          := _AxisRef, 
                  Execute       := FALSE);

  nState                        := 0;
END_IF

fActivePosition                 := fUsedPos;
MoveAbsolute                    := res;
END_METHOD

METHOD MoveEndless : ST_McOutputs
VAR_INPUT
  Execute       : BOOL;
  Position      : LREAL;
  Velocity      : LREAL;
  Acceleration  : LREAL;
  Deceleration  : LREAL;
  Jerk          : LREAL;
  BufferMode    : Tc2_MC2.MC_BufferMode;
END_VAR
VAR_INST
  diState       : DINT;
  rtrigErr      : Tc2_Standard.R_TRIG;
  res           : Tc2_MC2.ST_McOutputs;
  nAcc, nDec    : LREAL;
END_VAR

IF NOT Execute
THEN
  memset(ADR(res), 0, SIZEOF(res));
  diState := 0;
END_IF

CASE diState OF

  0:
    nAcc := SEL((Acceleration < 1.0), Acceleration,stDefaultAcceleration.fValue);
    nDec := SEL((Deceleration < 1.0), Deceleration,stDefaultDeceleration.fValue);

    IF (Position > 0)
    THEN
      fbMoveEndless.Position := Position + SQRT(nAcc)/(_rCycleTime*10_000);
    ELSE
      fbMoveEndless.Position := Position - SQRT(nAcc)/(_rCycleTime*10_000);
    END_IF

    fbMoveEndless(
      Axis            := _AxisRef, 
      Execute         := FALSE, 
      Velocity        := Velocity,
      EndVelocity     := Velocity, 
      Acceleration    := nAcc, 
      Deceleration    := nDec, 
      Jerk            := Jerk, 
      BufferMode      := BufferMode, 
      Options:= );

    IF NOT (Velocity > 0)
    THEN
      res.ErrorID     := 333;
      diState         := 99;

    ELSIF Execute
    THEN
      res.Busy        := TRUE;
      diState         := 10;
    END_IF
END_CASE

CASE diState OF
  10:
    fbMoveEndless(
      Axis          := _AxisRef, 
      Execute       := TRUE);


    IF fbMoveEndless.Error
    THEN
      res.ErrorID   := fbMoveEndless.ErrorID;

      // write list entry
      stMsg.eType           := E_MessageType.eMessageError;
      stMsg.eDevice         := e_Device.Axis + TO_DINT(_AxisRef.NcToPlc.AxisId);
      stMsg.eSubdevice      := e_SubDevice.fbMoveEndless;
      stMsg.iErrorNumber    := fbMoveEndless.ErrorID;
      f_MessageSet(stMsg);
      MsgAdd(stMsg);

      fbMoveEndless(
        Axis        := _AxisRef, 
        Execute     := FALSE);

      diState       := 99;

    ELSIF fbMoveEndless.InEndVelocity
    THEN
      fbMoveEndless(
        Axis        := _AxisRef, 
        Execute     := FALSE);

      diState       := 20;
    END_IF
END_CASE

CASE diState OF
  20:
    res.Error       := FALSE;
    res.Busy        := FALSE;
    res.Done        := TRUE;

  99:
    res.Error       := TRUE;
    res.Busy        := FALSE;
    res.Done        := FALSE;

END_CASE

MoveEndless := res;
END_METHOD

METHOD MovePtP : ST_McOutputs
VAR_INPUT
  (* HAUD 2022 03 23 *)
  (* trigger *)
  {attribute '''NORMAL__COMMENT' := ' trigger movement '}
  Execute : BOOL;
  (* Absolute target position to be used for positioning *)
  {attribute '''NORMAL__COMMENT' := ' Absolute target position to be used for positioning '}
  Position  : LREAL;
  (* Maximum travel velocity. If not specified, DefaultVelocity will be used *)
  {attribute '''NORMAL__COMMENT' := ' Maximum travel velocity. If not specified, DefaultVelocity will be used '}
  Velocity  : LREAL;
  (* Acceleration. If not specified, DefaultAcceleration will be used *)
  {attribute '''NORMAL__COMMENT' := ' Acceleration. If not specified, DefaultAcceleration will be used '}
  Acceleration  : LREAL;
  (* Deceleration. If not specified, DefaultDeceleration will be used *)
  {attribute '''NORMAL__COMMENT' := ' Deceleration. If not specified, DefaultDeceleration will be used '}
  Deceleration  : LREAL;
  (* Jerk. If not specified, DefaultJerk will be used *)
  {attribute '''NORMAL__COMMENT' := ' Jerk. If not specified, DefaultJerk will be used '}
  Jerk  : LREAL;
END_VAR
VAR_INST

  _nState   : DINT;
  _res      : ST_McOutputs;
  _stMsg    : ST_Message;
  _fbMove   : Tc2_MC2.MC_MoveAbsolute;
END_VAR

CASE _nState OF
  0:
    IF Execute
    THEN
      memset(ADR(_res), 0, SIZEOF(_res));

      _res.Busy                 := TRUE;

      _fbMove(Axis              := _AxisRef, 
              Execute           := FALSE, 
              Position          := Position, 
              Velocity          := Velocity, 
              Acceleration      := Acceleration, 
              Deceleration      := Deceleration, 
              Jerk              := Jerk, 
              BufferMode        := Tc2_MC2.MC_BufferMode.MC_Aborting);

      _nState                   := 10;
    END_IF
END_CASE
CASE _nState OF
  10:
    _fbMove(Axis                := _AxisRef, 
            Execute             := TRUE, 
            Position            := Position, 
            Velocity            := Velocity, 
            Acceleration        := Acceleration, 
            Deceleration        := Deceleration, 
            Jerk                := Jerk, 
            BufferMode          := Tc2_MC2.MC_BufferMode.MC_Aborting);

    IF _fbMove.Busy
    THEN
      _nState                   := 20;
    END_IF
END_CASE
CASE _nState OF
  20:
    _fbMove(Axis                := _AxisRef);

    IF NOT _fbMove.Error AND 
       NOT _AxisRef.Status.Error
    THEN
      IF _fbMove.Done
      THEN
        _nState                 := 30;
      END_IF
    ELSE
      _stMsg.eType              := E_MessageType.eMessageError;
      _stMsg.eDevice            := e_Device.Axis + TO_DINT(_AxisRef.NcToPlc.AxisId);
      _stMsg.eSubdevice         :=  e_SubDevice.fbMovePtP;
      _stMsg.iErrorNumber       := _fbMove.ErrorID;

      f_MessageSet(_stMsg);
      MsgAdd(_stMsg);

     _res.ErrorID               := _fbMove.ErrorID;

      _fbMove(Axis              := _AxisRef, 
             Execute            := FALSE);

      _nState                   := 99;
    END_IF
END_CASE
CASE _nState OF
  30:
    _res.Busy                   := FALSE;
    _res.Done                   := TRUE;

  99:
    _res.Busy                   := FALSE;
    _res.Error                  := TRUE;
END_CASE

IF NOT Execute
THEN
  memset(ADR(_res), 0, SIZEOF(_res));
  _nState                       := 0;
END_IF

MovePtP := _res;
END_METHOD

{attribute '''NORMAL__COMMENT' := ' MoveVelocity starts a continuous movement with specified velocity and direction. The movement can be stopped through an other travel command. Refer to MC_MoveVelocity Function Block
  in the Tc2_MC2 library; In Velocity will be indicated by the return value member Done. To instances of MC_MoveVelocity are used to trigger new parameter during movement '}
(* MoveVelocity starts a continuous movement with specified velocity and direction. The movement can be stopped through an other travel command. Refer to MC_MoveVelocity Function Block
  in the Tc2_MC2 library; In Velocity will be indicated by the return value member Done. To instances of MC_MoveVelocity are used to trigger new parameter during movement *)
METHOD MoveVelocity : Tc2_MC2.ST_McOutputs
VAR_INPUT
  Enable   : BOOL;
  (* Maximum travel velocity. If not specified, DefaultVelocity will be used *)
  {attribute '''NORMAL__COMMENT' := ' Maximum travel velocity. If not specified, DefaultVelocity will be used '}
  Velocity  : LREAL;
  (* Acceleration. If not specified, DefaultAcceleration will be used *)
  {attribute '''NORMAL__COMMENT' := ' Acceleration. If not specified, DefaultAcceleration will be used '}
  Acceleration  : LREAL;
  (* Deceleration. If not specified, DefaultDeceleration will be used *)
  {attribute '''NORMAL__COMMENT' := ' Deceleration. If not specified, DefaultDeceleration will be used '}
  Deceleration  : LREAL;
  (* Jerk. If not specified, DefaultJerk will be used *)
  {attribute '''NORMAL__COMMENT' := ' Jerk. If not specified, DefaultJerk will be used '}
  Jerk  : LREAL;
  (* direction of travel: MC_Positive_Direction, MC_Shortest_Way, MC_Negative_Direction, MC_Current_Direction *)
  {attribute '''NORMAL__COMMENT' := ' direction of travel: MC_Positive_Direction, MC_Shortest_Way, MC_Negative_Direction, MC_Current_Direction '}
  Direction : Tc2_MC2.MC_Direction := MC_Positive_Direction;
  (* The BufferMode is analyzed, if the axis is already executing another command. The running command can be aborted,
                    or the new command becomes active after the running command. The BufferMode also determines the transition condition from the current to the next command.
                    If the command is applied to a coupled slave axis used, the only available buffer mode is Aborting. *)
  {attribute '''NORMAL__COMMENT' := ' The BufferMode is analyzed, if the axis is already executing another command. The running command can be aborted,
                    or the new command becomes active after the running command. The BufferMode also determines the transition condition from the current to the next command.
                    If the command is applied to a coupled slave axis used, the only available buffer mode is Aborting. '}
  BufferMode  : Tc2_MC2.MC_BufferMode;
END_VAR
VAR_IN_OUT
  fActiveVelocity   : LREAL;
  eState            : e_AxisFunction;
END_VAR
VAR_INST
  res       : Tc2_MC2.ST_McOutputs;
  nState    : DINT;
  fUsedPos,
  fUsedVel,
  fUsedAcc,
  fUsedDec,
  fUsedJrk    : LREAL;
END_VAR
// Select Default values of dynamic parameter if 0 is specified
fUsedVel := Velocity;
fUsedAcc := Acceleration;
fUsedDec := Deceleration;
fUsedJrk := Jerk;

CASE nState OF
  0:
    IF Enable
    THEN
      memset(ADR(res),0,SIZEOF(res));

      res.Busy                      := TRUE;

      fUsedVel                      := SEL((Velocity < 0.01),Velocity, fDefaultVelocity);

      fbMoveVelocity1(Axis          := _AxisRef, 
                      Execute       := FALSE, 
                      Velocity      := fUsedVel, 
                      Acceleration  := fUsedAcc, 
                      Deceleration  := fUsedDec, 
                      Jerk          := fUsedJrk, 
                      Direction     := Direction, 
                      BufferMode    := BufferMode);

      fbMoveVelocity2(Axis          := _AxisRef, 
                      Execute       := FALSE, 
                      Acceleration  := fUsedAcc, 
                      Deceleration  := fUsedDec, 
                      Jerk          := fUsedJrk, 
                      Direction     := Direction, 
                      BufferMode    := BufferMode);

      nState                        := 10;
    END_IF
END_CASE
CASE nState OF
  10:
    eState                          := AXIS_BUSY;
    fbMoveVelocity1(Axis            := _AxisRef, 
                    Execute         := TRUE, 
                    Velocity        := fUsedVel, 
                    Acceleration    := fUsedAcc, 
                    Deceleration    := fUsedDec, 
                    Jerk            := fUsedJrk, 
                    Direction       := Direction, 
                    BufferMode      := BufferMode);

    IF fbMoveVelocity1.Error
    THEN
      stMsg.eType                   := E_MessageType.eMessageError;
      stMsg.eDevice                 := e_Device.Axis + TO_DINT(_AxisRef.NcToPlc.AxisId);
      stMsg.eSubdevice              := e_SubDevice.fbMoveVelocity1;
      stMsg.iErrorNumber            := fbMoveVelocity1.ErrorID;

      f_MessageSet(stMsg);
      MsgAdd(stMsg);

      res.ErrorID                   := fbMoveVelocity1.ErrorID;

      nState                        := 99;

    ELSIF fbMoveVelocity1.Active
    THEN
      res.Active                    := TRUE;
      nState                        := 20;
    END_IF
END_CASE
CASE nState OF
  20:
    fbMoveVelocity1(Axis            := _AxisRef);
    fbMoveVelocity2(Axis            := _AxisRef);

    res.Done                        := fbMoveVelocity1.InVelocity;

    IF fbMoveVelocity1.Error
    THEN
      stMsg.eType                   := E_MessageType.eMessageError;
      stMsg.eDevice                 := e_Device.Axis + TO_DINT(_AxisRef.NcToPlc.AxisId);
      stMsg.eSubdevice              := e_SubDevice.fbMoveVelocity1;
      stMsg.iErrorNumber            := fbMoveVelocity1.ErrorID;

      f_MessageSet(stMsg);
      MsgAdd(stMsg);

      res.ErrorID                   := fbMoveVelocity1.ErrorID;

      nState                        := 99;


    ELSIF (Velocity <> fUsedVel)
    THEN

      fUsedVel                      := SEL((Velocity < 0.01),Velocity, fDefaultVelocity);

    fbMoveVelocity1(Axis            := _AxisRef, 
                    Execute         := FALSE);

      fbMoveVelocity2(Axis          := _AxisRef, 
                      Execute       := TRUE, 
                      Velocity      := fUsedVel, 
                      Acceleration  := fUsedAcc, 
                      Deceleration  := fUsedDec, 
                      Jerk          := fUsedJrk, 
                      Direction     := Direction, 
                      BufferMode    := BufferMode);

      nState                        := 30;
    END_IF
END_CASE
CASE nState OF
  30:
    eState                          := AXIS_ACK;
    fbMoveVelocity1(Axis            := _AxisRef);
    fbMoveVelocity2(Axis            := _AxisRef);

    res.Done                        := fbMoveVelocity2.InVelocity;

    IF fbMoveVelocity2.Error
    THEN
      stMsg.eType                   := E_MessageType.eMessageError;
      stMsg.eDevice                 := e_Device.Axis + UDINT_TO_DINT(_AxisRef.NcToPlc.AxisId);
      stMsg.eSubdevice              := e_SubDevice.fbMoveVelocity2;
      stMsg.iErrorNumber            := fbMoveVelocity2.ErrorID;

      f_MessageSet(stMsg);
      MsgAdd(stMsg);

      res.ErrorID                   := fbMoveVelocity2.ErrorID;

      nState                        := 99;

    ELSIF fbMoveVelocity2.InVelocity
    THEN
      nState                        := 40;
    END_IF
END_CASE
CASE nState OF
  40:
    fbMoveVelocity1(Axis            := _AxisRef);
    fbMoveVelocity2(Axis            := _AxisRef);

    res.Done                        := fbMoveVelocity2.InVelocity;

    IF fbMoveVelocity2.Error
    THEN
      stMsg.eType                   := E_MessageType.eMessageError;
      stMsg.eDevice                 := e_Device.Axis + UDINT_TO_DINT(_AxisRef.NcToPlc.AxisId);
      stMsg.eSubdevice              := e_SubDevice.fbMoveVelocity2;
      stMsg.iErrorNumber            := fbMoveVelocity2.ErrorID;

      f_MessageSet(stMsg);
      MsgAdd(stMsg);

      res.ErrorID                   := fbMoveVelocity2.ErrorID;

      nState                        := 99;

    ELSIF (Velocity <> fUsedVel)
    THEN
      nState                        := 10;
      fbMoveVelocity2(Axis          := _AxisRef, 
                    Execute         := FALSE);
    END_IF
END_CASE

CASE nState OF
  99:
    res.Busy                        := FALSE;
    res.Done                        := FALSE;
    res.Error                       := TRUE;
END_CASE


IF NOT Enable
THEN
  eState                            := AXIS_DISABLE;
  fUsedVel                          := 0.0;
  memset(ADR(res),0,SIZEOF(res));
  fbMoveVelocity1(Axis              := _AxisRef, 
                  Execute           := FALSE);

  fbMoveVelocity2(Axis              := _AxisRef, 
                  Execute           := FALSE);
 
  nState                            := 0;
END_IF

fActiveVelocity := fUsedVel;
MoveVelocity := res;
END_METHOD

METHOD MsgAdd : BOOL
VAR_INPUT
  stMsg : ST_Message;
END_VAR

atMsg[itMsg] := stMsg;
itMsg := itMsg + 1;
itMsg := SEL((itMsg > MAX_MSG_INTERN),itMsg,1);
END_METHOD

